ABB RAPID module: P61.mod

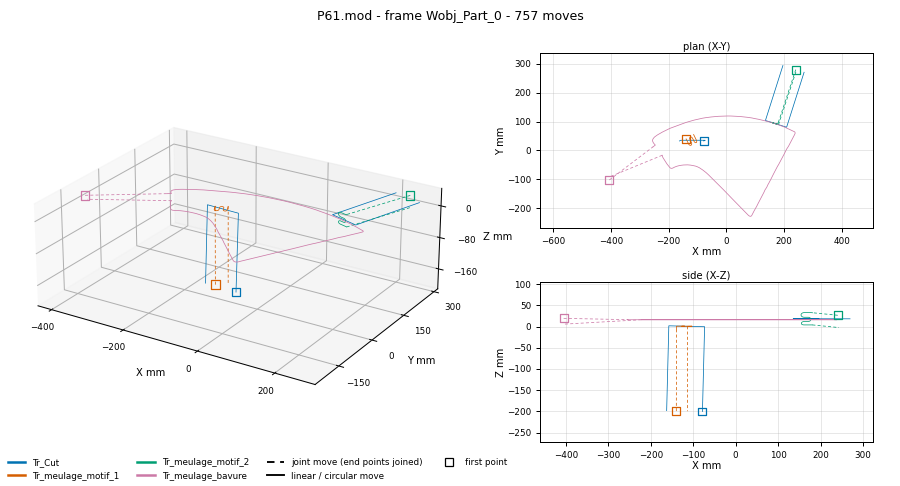
[picture p0: tool path of P61.mod in frame Wobj_Part_0, 757 of 767 moves have a stored position in this frame; points joined in program order, loops and branches not executed]
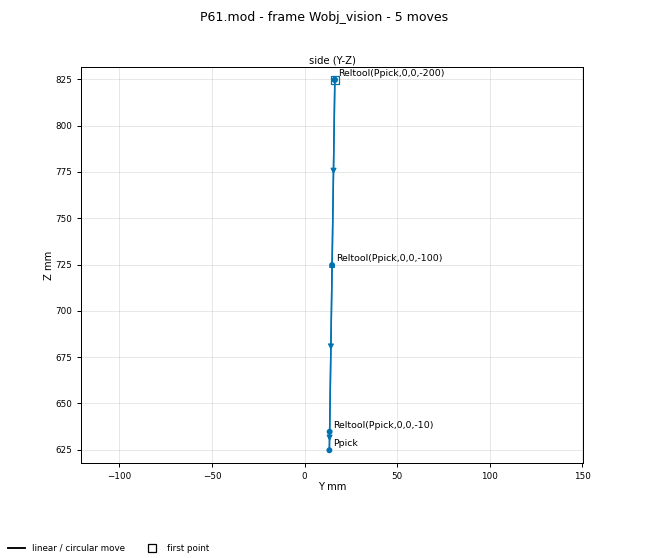
[picture p1: tool path of P61.mod in frame Wobj_vision, 5 of 767 moves have a stored position in this frame; points joined in program order, loops and branches not executed]
MODULE P61
	LOCAL CONST Speeddata vitesse_Tronconnage :=[10, 500, 0, 0];
	LOCAL CONST Robtarget Coupe_0 :=[[-120.4273984375,35.4203203125,0.733973022460938],[0.716031512015104,-0.00434153413134131,-0.698040250859739,0.00445343265621212],[0,0,0,0],[8.999999E+09,8.999999E+09,8.999999E+09,8.999999E+09,8.999999E+09,8.999999E+09]];
	LOCAL CONST Robtarget Coupe_1 :=[[167.499296875,93.7912890625,18.2855390625],[0.417597748453561,0.417256329208566,-0.570874027904049,-0.570624325179462],[0,0,0,0],[8.999999E+09,8.999999E+09,8.999999E+09,8.999999E+09,8.999999E+09,8.999999E+09]];
	LOCAL CONST Robtarget Tr_meulage_motif_1_App1 :=[[-139.92964037527,40.0496042134107,-199.309536992709],[-7.8362214742082E-08,0.00132363335464177,5.92023053405581E-05,0.999999122244526],[0,0,0,0],[8.999999E+09,8.999999E+09,8.999999E+09,8.999999E+09,8.999999E+09,8.999999E+09]];
	LOCAL CONST Robtarget Tr_meulage_motif_1_App2 :=[[-139.426660143764,40.072101109108,-9.31020408657393],[-7.8362214742082E-08,0.00132363335464177,5.92023053405581E-05,0.999999122244526],[0,0,0,0],[8.999999E+09,8.999999E+09,8.999999E+09,8.999999E+09,8.999999E+09,8.999999E+09]];
	LOCAL CONST Robtarget Tr_meulage_motif_1_P0 :=[[-139.4001875,40.07328515625,0.689760803222656],[-7.8362214742082E-08,0.00132363335464177,5.92023053405581E-05,0.999999122244526],[0,0,0,0],[8.999999E+09,8.999999E+09,8.999999E+09,8.999999E+09,8.999999E+09,8.999999E+09]];
	LOCAL CONST Robtarget Tr_meulage_motif_1_P1 :=[[-138.96090625,39.1750078125,0.700619750976562],[-7.8362214742082E-08,0.00132363335464177,5.92023053405581E-05,0.999999122244526],[0,0,0,0],[8.999999E+09,8.999999E+09,8.999999E+09,8.999999E+09,8.999999E+09,8.999999E+09]];
	LOCAL CONST Robtarget Tr_meulage_motif_1_P2 :=[[-138.521609375,38.27673046875,0.711478759765625],[-7.8362214742082E-08,0.00132363335464177,5.92023053405581E-05,0.999999122244526],[0,0,0,0],[8.999999E+09,8.999999E+09,8.999999E+09,8.999999E+09,8.999999E+09,8.999999E+09]];
	LOCAL CONST Robtarget Tr_meulage_motif_1_P3 :=[[-138.0823125,37.378453125,0.722337707519531],[-7.8362214742082E-08,0.00132363335464177,5.92023053405581E-05,0.999999122244526],[0,0,0,0],[8.999999E+09,8.999999E+09,8.999999E+09,8.999999E+09,8.999999E+09,8.999999E+09]];
	LOCAL CONST Robtarget Tr_meulage_motif_1_P4 :=[[-137.643015625,36.480171875,0.733196716308594],[-7.8362214742082E-08,0.00132363335464177,5.92023053405581E-05,0.999999122244526],[0,0,0,0],[8.999999E+09,8.999999E+09,8.999999E+09,8.999999E+09,8.999999E+09,8.999999E+09]];
	LOCAL CONST Robtarget Tr_meulage_motif_1_P5 :=[[-137.203734375,35.58189453125,0.744055725097656],[-7.8362214742082E-08,0.00132363335464177,5.92023053405581E-05,0.999999122244526],[0,0,0,0],[8.999999E+09,8.999999E+09,8.999999E+09,8.999999E+09,8.999999E+09,8.999999E+09]];
	LOCAL CONST Robtarget Tr_meulage_motif_1_P6 :=[[-136.7644375,34.6836171875,0.754914672851563],[-7.8362214742082E-08,0.00132363335464177,5.92023053405581E-05,0.999999122244526],[0,0,0,0],[8.999999E+09,8.999999E+09,8.999999E+09,8.999999E+09,8.999999E+09,8.999999E+09]];
	LOCAL CONST Robtarget Tr_meulage_motif_1_P7 :=[[-136.325140625,33.78533984375,0.765773681640625],[-7.8362214742082E-08,0.00132363335464177,5.92023053405581E-05,0.999999122244526],[0,0,0,0],[8.999999E+09,8.999999E+09,8.999999E+09,8.999999E+09,8.999999E+09,8.999999E+09]];
	LOCAL CONST Robtarget Tr_meulage_motif_1_P8 :=[[-135.88584375,32.88705859375,0.776632629394531],[-7.8362214742082E-08,0.00132363335464177,5.92023053405581E-05,0.999999122244526],[0,0,0,0],[8.999999E+09,8.999999E+09,8.999999E+09,8.999999E+09,8.999999E+09,8.999999E+09]];
	LOCAL CONST Robtarget Tr_meulage_motif_1_P9 :=[[-135.4465625,31.98878125,0.787491638183594],[-7.8362214742082E-08,0.00132363335464177,5.92023053405581E-05,0.999999122244526],[0,0,0,0],[8.999999E+09,8.999999E+09,8.999999E+09,8.999999E+09,8.999999E+09,8.999999E+09]];
	LOCAL CONST Robtarget Tr_meulage_motif_1_P10 :=[[-135.007265625,31.09050390625,0.7983505859375],[-7.8362214742082E-08,0.00132363335464177,5.92023053405581E-05,0.999999122244526],[0,0,0,0],[8.999999E+09,8.999999E+09,8.999999E+09,8.999999E+09,8.999999E+09,8.999999E+09]];
	LOCAL CONST Robtarget Tr_meulage_motif_1_P11 :=[[-134.56796875,30.192224609375,0.809209594726563],[-7.8362214742082E-08,0.00132363335464177,5.92023053405581E-05,0.999999122244526],[0,0,0,0],[8.999999E+09,8.999999E+09,8.999999E+09,8.999999E+09,8.999999E+09,8.999999E+09]];
	LOCAL CONST Robtarget Tr_meulage_motif_1_P12 :=[[-134.128671875,29.293947265625,0.820068603515625],[-7.8362214742082E-08,0.00132363335464177,5.92023053405581E-05,0.999999122244526],[0,0,0,0],[8.999999E+09,8.999999E+09,8.999999E+09,8.999999E+09,8.999999E+09,8.999999E+09]];
	LOCAL CONST Robtarget Tr_meulage_motif_1_P13 :=[[-133.689390625,28.39566796875,0.830927551269531],[-7.8362214742082E-08,0.00132363335464177,5.92023053405581E-05,0.999999122244526],[0,0,0,0],[8.999999E+09,8.999999E+09,8.999999E+09,8.999999E+09,8.999999E+09,8.999999E+09]];
	LOCAL CONST Robtarget Tr_meulage_motif_1_P14 :=[[-133.25009375,27.497390625,0.841786560058594],[-7.8362214742082E-08,0.00132363335464177,5.92023053405581E-05,0.999999122244526],[0,0,0,0],[8.999999E+09,8.999999E+09,8.999999E+09,8.999999E+09,8.999999E+09,8.999999E+09]];
	LOCAL CONST Robtarget Tr_meulage_motif_1_P15 :=[[-132.810796875,26.599111328125,0.8526455078125],[-7.8362214742082E-08,0.00132363335464177,5.92023053405581E-05,0.999999122244526],[0,0,0,0],[8.999999E+09,8.999999E+09,8.999999E+09,8.999999E+09,8.999999E+09,8.999999E+09]];
	LOCAL CONST Robtarget Tr_meulage_motif_1_P16 :=[[-132.371515625,25.700833984375,0.863504516601562],[-7.8362214742082E-08,0.00132363335464177,5.92023053405581E-05,0.999999122244526],[0,0,0,0],[8.999999E+09,8.999999E+09,8.999999E+09,8.999999E+09,8.999999E+09,8.999999E+09]];
	LOCAL CONST Robtarget Tr_meulage_motif_1_P17 :=[[-131.93221875,24.8025546875,0.874363525390625],[-7.8362214742082E-08,0.00132363335464177,5.92023053405581E-05,0.999999122244526],[0,0,0,0],[8.999999E+09,8.999999E+09,8.999999E+09,8.999999E+09,8.999999E+09,8.999999E+09]];
	LOCAL CONST Robtarget Tr_meulage_motif_1_P18 :=[[-131.492921875,23.90427734375,0.885222473144531],[-7.8362214742082E-08,0.00132363335464177,5.92023053405581E-05,0.999999122244526],[0,0,0,0],[8.999999E+09,8.999999E+09,8.999999E+09,8.999999E+09,8.999999E+09,8.999999E+09]];
	LOCAL CONST Robtarget Tr_meulage_motif_1_P19 :=[[-131.0536328125,23.005998046875,0.896081481933594],[-7.8362214742082E-08,0.00132363335464177,5.92023053405581E-05,0.999999122244526],[0,0,0,0],[8.999999E+09,8.999999E+09,8.999999E+09,8.999999E+09,8.999999E+09,8.999999E+09]];
	LOCAL CONST Robtarget Tr_meulage_motif_1_P20 :=[[-130.6143359375,22.107720703125,0.9069404296875],[-7.8362214742082E-08,0.00132363335464177,5.92023053405581E-05,0.999999122244526],[0,0,0,0],[8.999999E+09,8.999999E+09,8.999999E+09,8.999999E+09,8.999999E+09,8.999999E+09]];
	LOCAL CONST Robtarget Tr_meulage_motif_1_P21 :=[[-130.0789609375,21.264701171875,0.917042663574219],[-7.8362214742082E-08,0.00132363335464177,5.92023053405581E-05,0.999999122244526],[0,0,0,0],[8.999999E+09,8.999999E+09,8.999999E+09,8.999999E+09,8.999999E+09,8.999999E+09]];
	LOCAL CONST Robtarget Tr_meulage_motif_1_P22 :=[[-129.473453125,20.507244140625,0.926029846191406],[-7.8362214742082E-08,0.00132363335464177,5.92023053405581E-05,0.999999122244526],[0,0,0,0],[8.999999E+09,8.999999E+09,8.999999E+09,8.999999E+09,8.999999E+09,8.999999E+09]];
	LOCAL CONST Robtarget Tr_meulage_motif_1_P23 :=[[-128.8546484375,19.860673828125,0.9336279296875],[-7.8362214742082E-08,0.00132363335464177,5.92023053405581E-05,0.999999122244526],[0,0,0,0],[8.999999E+09,8.999999E+09,8.999999E+09,8.999999E+09,8.999999E+09,8.999999E+09]];
	LOCAL CONST Robtarget Tr_meulage_motif_1_P24 :=[[-128.2773203125,19.3082265625,0.940084838867188],[-7.8362214742082E-08,0.00132363335464177,5.92023053405581E-05,0.999999122244526],[0,0,0,0],[8.999999E+09,8.999999E+09,8.999999E+09,8.999999E+09,8.999999E+09,8.999999E+09]];
	LOCAL CONST Robtarget Tr_meulage_motif_1_P25 :=[[-127.240140625,18.589798828125,0.948275268554687],[-7.8362214742082E-08,0.00132363335464177,5.92023053405581E-05,0.999999122244526],[0,0,0,0],[8.999999E+09,8.999999E+09,8.999999E+09,8.999999E+09,8.999999E+09,8.999999E+09]];
	LOCAL CONST Robtarget Tr_meulage_motif_1_P26 :=[[-126.028875,18.042408203125,0.954212341308594],[-7.8362214742082E-08,0.00132363335464177,5.92023053405581E-05,0.999999122244526],[0,0,0,0],[8.999999E+09,8.999999E+09,8.999999E+09,8.999999E+09,8.999999E+09,8.999999E+09]];
	LOCAL CONST Robtarget Tr_meulage_motif_1_P27 :=[[-124.7367109375,17.73071484375,0.957158752441406],[-7.8362214742082E-08,0.00132363335464177,5.92023053405581E-05,0.999999122244526],[0,0,0,0],[8.999999E+09,8.999999E+09,8.999999E+09,8.999999E+09,8.999999E+09,8.999999E+09]];
	LOCAL CONST Robtarget Tr_meulage_motif_1_P28 :=[[-123.519546875,17.782501953125,0.955637145996094],[-7.8362214742082E-08,0.00132363335464177,5.92023053405581E-05,0.999999122244526],[0,0,0,0],[8.999999E+09,8.999999E+09,8.999999E+09,8.999999E+09,8.999999E+09,8.999999E+09]];
	LOCAL CONST Robtarget Tr_meulage_motif_1_P29 :=[[-122.8824375,18.063896484375,0.951677001953125],[-7.8362214742082E-08,0.00132363335464177,5.92023053405581E-05,0.999999122244526],[0,0,0,0],[8.999999E+09,8.999999E+09,8.999999E+09,8.999999E+09,8.999999E+09,8.999999E+09]];
	LOCAL CONST Robtarget Tr_meulage_motif_1_P30 :=[[-122.28840625,18.3543515625,0.947635192871094],[-7.8362214742082E-08,0.00132363335464177,5.92023053405581E-05,0.999999122244526],[0,0,0,0],[8.999999E+09,8.999999E+09,8.999999E+09,8.999999E+09,8.999999E+09,8.999999E+09]];
	LOCAL CONST Robtarget Tr_meulage_motif_1_P31 :=[[-121.718625,18.69403125,0.942998474121094],[-7.8362214742082E-08,0.00132363335464177,5.92023053405581E-05,0.999999122244526],[0,0,0,0],[8.999999E+09,8.999999E+09,8.999999E+09,8.999999E+09,8.999999E+09,8.999999E+09]];
	LOCAL CONST Robtarget Tr_meulage_motif_1_P32 :=[[-120.9477421875,19.625513671875,0.930854064941406],[-7.8362214742082E-08,0.00132363335464177,5.92023053405581E-05,0.999999122244526],[0,0,0,0],[8.999999E+09,8.999999E+09,8.999999E+09,8.999999E+09,8.999999E+09,8.999999E+09]];
	LOCAL CONST Robtarget Tr_meulage_motif_1_P33 :=[[-120.4197578125,20.837162109375,0.915399108886719],[-7.8362214742082E-08,0.00132363335464177,5.92023053405581E-05,0.999999122244526],[0,0,0,0],[8.999999E+09,8.999999E+09,8.999999E+09,8.999999E+09,8.999999E+09,8.999999E+09]];
	LOCAL CONST Robtarget Tr_meulage_motif_1_P34 :=[[-120.1247109375,22.12055078125,0.899219604492188],[-7.8362214742082E-08,0.00132363335464177,5.92023053405581E-05,0.999999122244526],[0,0,0,0],[8.999999E+09,8.999999E+09,8.999999E+09,8.999999E+09,8.999999E+09,8.999999E+09]];
	LOCAL CONST Robtarget Tr_meulage_motif_1_P35 :=[[-120.07103125,22.9115859375,0.889339538574219],[-7.8362214742082E-08,0.00132363335464177,5.92023053405581E-05,0.999999122244526],[0,0,0,0],[8.999999E+09,8.999999E+09,8.999999E+09,8.999999E+09,8.999999E+09,8.999999E+09]];
	LOCAL CONST Robtarget Tr_meulage_motif_1_P36 :=[[-120.141828125,24.166080078125,0.873783142089844],[-7.8362214742082E-08,0.00132363335464177,5.92023053405581E-05,0.999999122244526],[0,0,0,0],[8.999999E+09,8.999999E+09,8.999999E+09,8.999999E+09,8.999999E+09,8.999999E+09]];
	LOCAL CONST Robtarget Tr_meulage_motif_1_P37 :=[[-120.275796875,25.04115625,0.862992736816406],[-7.8362214742082E-08,0.00132363335464177,5.92023053405581E-05,0.999999122244526],[0,0,0,0],[8.999999E+09,8.999999E+09,8.999999E+09,8.999999E+09,8.999999E+09,8.999999E+09]];
	LOCAL CONST Robtarget Tr_meulage_motif_1_P38 :=[[-120.5015390625,25.968166015625,0.851622375488281],[-7.8362214742082E-08,0.00132363335464177,5.92023053405581E-05,0.999999122244526],[0,0,0,0],[8.999999E+09,8.999999E+09,8.999999E+09,8.999999E+09,8.999999E+09,8.999999E+09]];
	LOCAL CONST Robtarget Tr_meulage_motif_1_P39 :=[[-120.835171875,26.89758203125,0.840299865722656],[-7.8362214742082E-08,0.00132363335464177,5.92023053405581E-05,0.999999122244526],[0,0,0,0],[8.999999E+09,8.999999E+09,8.999999E+09,8.999999E+09,8.999999E+09,8.999999E+09]];
	LOCAL CONST Robtarget Tr_meulage_motif_1_P40 :=[[-121.1718515625,27.8377578125,0.828845642089844],[-7.8362214742082E-08,0.00132363335464177,5.92023053405581E-05,0.999999122244526],[0,0,0,0],[8.999999E+09,8.999999E+09,8.999999E+09,8.999999E+09,8.999999E+09,8.999999E+09]];
	LOCAL CONST Robtarget Tr_meulage_motif_1_P41 :=[[-121.611140625,28.73603515625,0.817986633300781],[-7.8362214742082E-08,0.00132363335464177,5.92023053405581E-05,0.999999122244526],[0,0,0,0],[8.999999E+09,8.999999E+09,8.999999E+09,8.999999E+09,8.999999E+09,8.999999E+09]];
	LOCAL CONST Robtarget Tr_meulage_motif_1_P42 :=[[-122.0504375,29.634314453125,0.807127685546875],[-7.8362214742082E-08,0.00132363335464177,5.92023053405581E-05,0.999999122244526],[0,0,0,0],[8.999999E+09,8.999999E+09,8.999999E+09,8.999999E+09,8.999999E+09,8.999999E+09]];
	LOCAL CONST Robtarget Tr_meulage_motif_1_P43 :=[[-122.4897265625,30.532591796875,0.796268676757813],[-7.8362214742082E-08,0.00132363335464177,5.92023053405581E-05,0.999999122244526],[0,0,0,0],[8.999999E+09,8.999999E+09,8.999999E+09,8.999999E+09,8.999999E+09,8.999999E+09]];
	LOCAL CONST Robtarget Tr_meulage_motif_1_P44 :=[[-122.9290234375,31.43087109375,0.785409729003906],[-7.8362214742082E-08,0.00132363335464177,5.92023053405581E-05,0.999999122244526],[0,0,0,0],[8.999999E+09,8.999999E+09,8.999999E+09,8.999999E+09,8.999999E+09,8.999999E+09]];
	LOCAL CONST Robtarget Tr_meulage_motif_1_P45 :=[[-123.3683125,32.3291484375,0.774550720214844],[-7.8362214742082E-08,0.00132363335464177,5.92023053405581E-05,0.999999122244526],[0,0,0,0],[8.999999E+09,8.999999E+09,8.999999E+09,8.999999E+09,8.999999E+09,8.999999E+09]];
	LOCAL CONST Robtarget Tr_meulage_motif_1_P46 :=[[-123.807609375,33.22742578125,0.763691711425781],[-7.8362214742082E-08,0.00132363335464177,5.92023053405581E-05,0.999999122244526],[0,0,0,0],[8.999999E+09,8.999999E+09,8.999999E+09,8.999999E+09,8.999999E+09,8.999999E+09]];
	LOCAL CONST Robtarget Tr_meulage_motif_1_P47 :=[[-124.2468984375,34.12570703125,0.752832763671875],[-7.8362214742082E-08,0.00132363335464177,5.92023053405581E-05,0.999999122244526],[0,0,0,0],[8.999999E+09,8.999999E+09,8.999999E+09,8.999999E+09,8.999999E+09,8.999999E+09]];
	LOCAL CONST Robtarget Tr_meulage_motif_1_P48 :=[[-124.6861953125,35.023984375,0.741973754882812],[-7.8362214742082E-08,0.00132363335464177,5.92023053405581E-05,0.999999122244526],[0,0,0,0],[8.999999E+09,8.999999E+09,8.999999E+09,8.999999E+09,8.999999E+09,8.999999E+09]];
	LOCAL CONST Robtarget Tr_meulage_motif_1_P49 :=[[-125.125484375,35.92226171875,0.731114807128906],[-7.8362214742082E-08,0.00132363335464177,5.92023053405581E-05,0.999999122244526],[0,0,0,0],[8.999999E+09,8.999999E+09,8.999999E+09,8.999999E+09,8.999999E+09,8.999999E+09]];
	LOCAL CONST Robtarget Tr_meulage_motif_1_P50 :=[[-125.56478125,36.8205390625,0.720255798339844],[-7.8362214742082E-08,0.00132363335464177,5.92023053405581E-05,0.999999122244526],[0,0,0,0],[8.999999E+09,8.999999E+09,8.999999E+09,8.999999E+09,8.999999E+09,8.999999E+09]];
	LOCAL CONST Robtarget Tr_meulage_motif_1_P51 :=[[-126.0040703125,37.7188203125,0.709396789550781],[-7.8362214742082E-08,0.00132363335464177,5.92023053405581E-05,0.999999122244526],[0,0,0,0],[8.999999E+09,8.999999E+09,8.999999E+09,8.999999E+09,8.999999E+09,8.999999E+09]];
	LOCAL CONST Robtarget Tr_meulage_motif_1_P52 :=[[-126.443359375,38.61709765625,0.698537841796875],[-7.8362214742082E-08,0.00132363335464177,5.92023053405581E-05,0.999999122244526],[0,0,0,0],[8.999999E+09,8.999999E+09,8.999999E+09,8.999999E+09,8.999999E+09,8.999999E+09]];
	LOCAL CONST Robtarget Tr_meulage_motif_1_P53 :=[[-126.7800390625,39.5572734375,0.687083618164062],[-7.8362214742082E-08,0.00132363335464177,5.92023053405581E-05,0.999999122244526],[0,0,0,0],[8.999999E+09,8.999999E+09,8.999999E+09,8.999999E+09,8.999999E+09,8.999999E+09]];
	LOCAL CONST Robtarget Tr_meulage_motif_1_P54 :=[[-127.006109375,40.5002578125,0.675514770507813],[-7.8362214742082E-08,0.00132363335464177,5.92023053405581E-05,0.999999122244526],[0,0,0,0],[8.999999E+09,8.999999E+09,8.999999E+09,8.999999E+09,8.999999E+09,8.999999E+09]];
	LOCAL CONST Robtarget Tr_meulage_motif_1_P55 :=[[-127.1364921875,41.38564453125,0.664593505859375],[-7.8362214742082E-08,0.00132363335464177,5.92023053405581E-05,0.999999122244526],[0,0,0,0],[8.999999E+09,8.999999E+09,8.999999E+09,8.999999E+09,8.999999E+09,8.999999E+09]];
	LOCAL CONST Robtarget Tr_meulage_motif_1_P56 :=[[-127.1758125,42.15837109375,0.655008239746094],[-7.8362214742082E-08,0.00132363335464177,5.92023053405581E-05,0.999999122244526],[0,0,0,0],[8.999999E+09,8.999999E+09,8.999999E+09,8.999999E+09,8.999999E+09,8.999999E+09]];
	LOCAL CONST Robtarget Tr_meulage_motif_1_P57 :=[[-127.0350703125,43.37862890625,0.639725280761719],[-7.8362214742082E-08,0.00132363335464177,5.92023053405581E-05,0.999999122244526],[0,0,0,0],[8.999999E+09,8.999999E+09,8.999999E+09,8.999999E+09,8.999999E+09,8.999999E+09]];
	LOCAL CONST Robtarget Tr_meulage_motif_1_P58 :=[[-126.62103125,44.58499609375,0.624418212890625],[-7.8362214742082E-08,0.00132363335464177,5.92023053405581E-05,0.999999122244526],[0,0,0,0],[8.999999E+09,8.999999E+09,8.999999E+09,8.999999E+09,8.999999E+09,8.999999E+09]];
	LOCAL CONST Robtarget Tr_meulage_motif_1_P59 :=[[-125.91634375,45.525015625,0.61221533203125],[-7.8362214742082E-08,0.00132363335464177,5.92023053405581E-05,0.999999122244526],[0,0,0,0],[8.999999E+09,8.999999E+09,8.999999E+09,8.999999E+09,8.999999E+09,8.999999E+09]];
	LOCAL CONST Robtarget Tr_meulage_motif_1_P60 :=[[-125.374765625,45.9955,0.605971557617187],[-7.8362214742082E-08,0.00132363335464177,5.92023053405581E-05,0.999999122244526],[0,0,0,0],[8.999999E+09,8.999999E+09,8.999999E+09,8.999999E+09,8.999999E+09,8.999999E+09]];
	LOCAL CONST Robtarget Tr_meulage_motif_1_P61 :=[[-124.71109375,46.3910703125,0.60057177734375],[-7.8362214742082E-08,0.00132363335464177,5.92023053405581E-05,0.999999122244526],[0,0,0,0],[8.999999E+09,8.999999E+09,8.999999E+09,8.999999E+09,8.999999E+09,8.999999E+09]];
	LOCAL CONST Robtarget Tr_meulage_motif_1_P62 :=[[-123.9900703125,46.669109375,0.596592895507812],[-7.8362214742082E-08,0.00132363335464177,5.92023053405581E-05,0.999999122244526],[0,0,0,0],[8.999999E+09,8.999999E+09,8.999999E+09,8.999999E+09,8.999999E+09,8.999999E+09]];
	LOCAL CONST Robtarget Tr_meulage_motif_1_P63 :=[[-122.81015625,46.779,0.594375244140625],[-7.8362214742082E-08,0.00132363335464177,5.92023053405581E-05,0.999999122244526],[0,0,0,0],[8.999999E+09,8.999999E+09,8.999999E+09,8.999999E+09,8.999999E+09,8.999999E+09]];
	LOCAL CONST Robtarget Tr_meulage_motif_1_P64 :=[[-122.1020078125,46.66409375,0.595294372558594],[-7.8362214742082E-08,0.00132363335464177,5.92023053405581E-05,0.999999122244526],[0,0,0,0],[8.999999E+09,8.999999E+09,8.999999E+09,8.999999E+09,8.999999E+09,8.999999E+09]];
	LOCAL CONST Robtarget Tr_meulage_motif_1_P65 :=[[-120.9153515625,46.25687890625,0.599505187988281],[-7.8362214742082E-08,0.00132363335464177,5.92023053405581E-05,0.999999122244526],[0,0,0,0],[8.999999E+09,8.999999E+09,8.999999E+09,8.999999E+09,8.999999E+09,8.999999E+09]];
	LOCAL CONST Robtarget Tr_meulage_motif_1_P66 :=[[-120.285875,45.9127578125,0.603332763671875],[-7.8362214742082E-08,0.00132363335464177,5.92023053405581E-05,0.999999122244526],[0,0,0,0],[8.999999E+09,8.999999E+09,8.999999E+09,8.999999E+09,8.999999E+09,8.999999E+09]];
	LOCAL CONST Robtarget Tr_meulage_motif_1_P67 :=[[-119.306,45.14755859375,0.612146423339844],[-7.8362214742082E-08,0.00132363335464177,5.92023053405581E-05,0.999999122244526],[0,0,0,0],[8.999999E+09,8.999999E+09,8.999999E+09,8.999999E+09,8.999999E+09,8.999999E+09]];
	LOCAL CONST Robtarget Tr_meulage_motif_1_P68 :=[[-118.677859375,44.53574609375,0.619305297851563],[-7.8362214742082E-08,0.00132363335464177,5.92023053405581E-05,0.999999122244526],[0,0,0,0],[8.999999E+09,8.999999E+09,8.999999E+09,8.999999E+09,8.999999E+09,8.999999E+09]];
	LOCAL CONST Robtarget Tr_meulage_motif_1_P69 :=[[-118.0847578125,43.78836328125,0.628176086425781],[-7.8362214742082E-08,0.00132363335464177,5.92023053405581E-05,0.999999122244526],[0,0,0,0],[8.999999E+09,8.999999E+09,8.999999E+09,8.999999E+09,8.999999E+09,8.999999E+09]];
	LOCAL CONST Robtarget Tr_meulage_motif_1_P70 :=[[-117.5560078125,42.95434765625,0.638171081542969],[-7.8362214742082E-08,0.00132363335464177,5.92023053405581E-05,0.999999122244526],[0,0,0,0],[8.999999E+09,8.999999E+09,8.999999E+09,8.999999E+09,8.999999E+09,8.999999E+09]];
	LOCAL CONST Robtarget Tr_meulage_motif_1_P71 :=[[-117.0206328125,42.111328125,0.648273315429687],[-7.8362214742082E-08,0.00132363335464177,5.92023053405581E-05,0.999999122244526],[0,0,0,0],[8.999999E+09,8.999999E+09,8.999999E+09,8.999999E+09,8.999999E+09,8.999999E+09]];
	LOCAL CONST Robtarget Tr_meulage_motif_1_P72 :=[[-116.58134375,41.21305078125,0.65913232421875],[-7.8362214742082E-08,0.00132363335464177,5.92023053405581E-05,0.999999122244526],[0,0,0,0],[8.999999E+09,8.999999E+09,8.999999E+09,8.999999E+09,8.999999E+09,8.999999E+09]];
	LOCAL CONST Robtarget Tr_meulage_motif_1_P73 :=[[-116.142046875,40.31476953125,0.669991333007813],[-7.8362214742082E-08,0.00132363335464177,5.92023053405581E-05,0.999999122244526],[0,0,0,0],[8.999999E+09,8.999999E+09,8.999999E+09,8.999999E+09,8.999999E+09,8.999999E+09]];
	LOCAL CONST Robtarget Tr_meulage_motif_1_P74 :=[[-115.7027578125,39.4164921875,0.680850280761719],[-7.8362214742082E-08,0.00132363335464177,5.92023053405581E-05,0.999999122244526],[0,0,0,0],[8.999999E+09,8.999999E+09,8.999999E+09,8.999999E+09,8.999999E+09,8.999999E+09]];
	LOCAL CONST Robtarget Tr_meulage_motif_1_P75 :=[[-115.2634609375,38.51821484375,0.691709289550781],[-7.8362214742082E-08,0.00132363335464177,5.92023053405581E-05,0.999999122244526],[0,0,0,0],[8.999999E+09,8.999999E+09,8.999999E+09,8.999999E+09,8.999999E+09,8.999999E+09]];
	LOCAL CONST Robtarget Tr_meulage_motif_1_P76 :=[[-114.824171875,37.6199375,0.702568237304688],[-7.8362214742082E-08,0.00132363335464177,5.92023053405581E-05,0.999999122244526],[0,0,0,0],[8.999999E+09,8.999999E+09,8.999999E+09,8.999999E+09,8.999999E+09,8.999999E+09]];
	LOCAL CONST Robtarget Tr_meulage_motif_1_P77 :=[[-114.384875,36.72165625,0.71342724609375],[-7.8362214742082E-08,0.00132363335464177,5.92023053405581E-05,0.999999122244526],[0,0,0,0],[8.999999E+09,8.999999E+09,8.999999E+09,8.999999E+09,8.999999E+09,8.999999E+09]];
	LOCAL CONST Robtarget Tr_meulage_motif_1_P78 :=[[-113.9455859375,35.82337890625,0.724286193847656],[-7.8362214742082E-08,0.00132363335464177,5.92023053405581E-05,0.999999122244526],[0,0,0,0],[8.999999E+09,8.999999E+09,8.999999E+09,8.999999E+09,8.999999E+09,8.999999E+09]];
	LOCAL CONST Robtarget Tr_meulage_motif_1_P79 :=[[-113.5062890625,34.9251015625,0.735145202636719],[-7.8362214742082E-08,0.00132363335464177,5.92023053405581E-05,0.999999122244526],[0,0,0,0],[8.999999E+09,8.999999E+09,8.999999E+09,8.999999E+09,8.999999E+09,8.999999E+09]];
	LOCAL CONST Robtarget Tr_meulage_motif_1_P80 :=[[-113.067,34.02682421875,0.746004211425781],[-7.8362214742082E-08,0.00132363335464177,5.92023053405581E-05,0.999999122244526],[0,0,0,0],[8.999999E+09,8.999999E+09,8.999999E+09,8.999999E+09,8.999999E+09,8.999999E+09]];
	LOCAL CONST Robtarget Tr_meulage_motif_1_P81 :=[[-112.627703125,33.12854296875,0.756863159179687],[-7.8362214742082E-08,0.00132363335464177,5.92023053405581E-05,0.999999122244526],[0,0,0,0],[8.999999E+09,8.999999E+09,8.999999E+09,8.999999E+09,8.999999E+09,8.999999E+09]];
	LOCAL CONST Robtarget Tr_meulage_motif_1_P82 :=[[-112.1884140625,32.230265625,0.76772216796875],[-7.8362214742082E-08,0.00132363335464177,5.92023053405581E-05,0.999999122244526],[0,0,0,0],[8.999999E+09,8.999999E+09,8.999999E+09,8.999999E+09,8.999999E+09,8.999999E+09]];
	LOCAL CONST Robtarget Tr_meulage_motif_1_P83 :=[[-111.7491171875,31.33198828125,0.778581115722656],[-7.8362214742082E-08,0.00132363335464177,5.92023053405581E-05,0.999999122244526],[0,0,0,0],[8.999999E+09,8.999999E+09,8.999999E+09,8.999999E+09,8.999999E+09,8.999999E+09]];
	LOCAL CONST Robtarget Tr_meulage_motif_1_P84 :=[[-111.2137421875,30.48896875,0.788683349609375],[-7.8362214742082E-08,0.00132363335464177,5.92023053405581E-05,0.999999122244526],[0,0,0,0],[8.999999E+09,8.999999E+09,8.999999E+09,8.999999E+09,8.999999E+09,8.999999E+09]];
	LOCAL CONST Robtarget Tr_meulage_motif_1_P85 :=[[-110.608234375,29.73151171875,0.797670532226562],[-7.8362214742082E-08,0.00132363335464177,5.92023053405581E-05,0.999999122244526],[0,0,0,0],[8.999999E+09,8.999999E+09,8.999999E+09,8.999999E+09,8.999999E+09,8.999999E+09]];
	LOCAL CONST Robtarget Tr_meulage_motif_1_P86 :=[[-109.9894296875,29.08494140625,0.805268615722656],[-7.8362214742082E-08,0.00132363335464177,5.92023053405581E-05,0.999999122244526],[0,0,0,0],[8.999999E+09,8.999999E+09,8.999999E+09,8.999999E+09,8.999999E+09,8.999999E+09]];
	LOCAL CONST Robtarget Tr_meulage_motif_1_P87 :=[[-109.4121015625,28.532494140625,0.811725524902344],[-7.8362214742082E-08,0.00132363335464177,5.92023053405581E-05,0.999999122244526],[0,0,0,0],[8.999999E+09,8.999999E+09,8.999999E+09,8.999999E+09,8.999999E+09,8.999999E+09]];
	LOCAL CONST Robtarget Tr_meulage_motif_1_P88 :=[[-108.374921875,27.81406640625,0.819916015625],[-7.8362214742082E-08,0.00132363335464177,5.92023053405581E-05,0.999999122244526],[0,0,0,0],[8.999999E+09,8.999999E+09,8.999999E+09,8.999999E+09,8.999999E+09,8.999999E+09]];
	LOCAL CONST Robtarget Tr_meulage_motif_1_P89 :=[[-107.16365625,27.26667578125,0.825853088378906],[-7.8362214742082E-08,0.00132363335464177,5.92023053405581E-05,0.999999122244526],[0,0,0,0],[8.999999E+09,8.999999E+09,8.999999E+09,8.999999E+09,8.999999E+09,8.999999E+09]];
	LOCAL CONST Robtarget Tr_meulage_motif_1_P90 :=[[-105.8764375,27.058552734375,0.827514526367187],[-7.8362214742082E-08,0.00132363335464177,5.92023053405581E-05,0.999999122244526],[0,0,0,0],[8.999999E+09,8.999999E+09,8.999999E+09,8.999999E+09,8.999999E+09,8.999999E+09]];
	LOCAL CONST Robtarget Tr_meulage_motif_1_P91 :=[[-104.7729765625,27.249388671875,0.824344848632813],[-7.8362214742082E-08,0.00132363335464177,5.92023053405581E-05,0.999999122244526],[0,0,0,0],[8.999999E+09,8.999999E+09,8.999999E+09,8.999999E+09,8.999999E+09,8.999999E+09]];
	LOCAL CONST Robtarget Tr_meulage_motif_1_P92 :=[[-104.2773125,27.557384765625,0.82015576171875],[-7.8362214742082E-08,0.00132363335464177,5.92023053405581E-05,0.999999122244526],[0,0,0,0],[8.999999E+09,8.999999E+09,8.999999E+09,8.999999E+09,8.999999E+09,8.999999E+09]];
	LOCAL CONST Robtarget Tr_meulage_motif_1_P93 :=[[-103.8999921875,27.737076171875,0.817648193359375],[-7.8362214742082E-08,0.00132363335464177,5.92023053405581E-05,0.999999122244526],[0,0,0,0],[8.999999E+09,8.999999E+09,8.999999E+09,8.999999E+09,8.999999E+09,8.999999E+09]];
	LOCAL CONST Robtarget Tr_meulage_motif_1_P94 :=[[-103.1883125,28.488166015625,0.807790771484375],[-7.8362214742082E-08,0.00132363335464177,5.92023053405581E-05,0.999999122244526],[0,0,0,0],[8.999999E+09,8.999999E+09,8.999999E+09,8.999999E+09,8.999999E+09,8.999999E+09]];
	LOCAL CONST Robtarget Tr_meulage_motif_1_P95 :=[[-102.7250078125,29.629576171875,0.79325634765625],[-7.8362214742082E-08,0.00132363335464177,5.92023053405581E-05,0.999999122244526],[0,0,0,0],[8.999999E+09,8.999999E+09,8.999999E+09,8.999999E+09,8.999999E+09,8.999999E+09]];
	LOCAL CONST Robtarget Tr_meulage_motif_1_P96 :=[[-102.613984375,30.36523828125,0.784023803710937],[-7.8362214742082E-08,0.00132363335464177,5.92023053405581E-05,0.999999122244526],[0,0,0,0],[8.999999E+09,8.999999E+09,8.999999E+09,8.999999E+09,8.999999E+09,8.999999E+09]];
	LOCAL CONST Robtarget Tr_meulage_motif_1_P97 :=[[-102.6340078125,31.613568359375,0.768507507324219],[-7.8362214742082E-08,0.00132363335464177,5.92023053405581E-05,0.999999122244526],[0,0,0,0],[8.999999E+09,8.999999E+09,8.999999E+09,8.999999E+09,8.999999E+09,8.999999E+09]];
	LOCAL CONST Robtarget Tr_meulage_motif_1_P98 :=[[-102.7679765625,32.48864453125,0.757717102050781],[-7.8362214742082E-08,0.00132363335464177,5.92023053405581E-05,0.999999122244526],[0,0,0,0],[8.999999E+09,8.999999E+09,8.999999E+09,8.999999E+09,8.999999E+09,8.999999E+09]];
	LOCAL CONST Robtarget Tr_meulage_motif_1_P99 :=[[-102.9937109375,33.41565234375,0.746346740722656],[-7.8362214742082E-08,0.00132363335464177,5.92023053405581E-05,0.999999122244526],[0,0,0,0],[8.999999E+09,8.999999E+09,8.999999E+09,8.999999E+09,8.999999E+09,8.999999E+09]];
	LOCAL CONST Robtarget Tr_meulage_motif_1_P100 :=[[-103.3273515625,34.3450703125,0.735024230957031],[-7.8362214742082E-08,0.00132363335464177,5.92023053405581E-05,0.999999122244526],[0,0,0,0],[8.999999E+09,8.999999E+09,8.999999E+09,8.999999E+09,8.999999E+09,8.999999E+09]];
	LOCAL CONST Robtarget Tr_meulage_motif_1_P101 :=[[-103.6640234375,35.28524609375,0.723570007324219],[-7.8362214742082E-08,0.00132363335464177,5.92023053405581E-05,0.999999122244526],[0,0,0,0],[8.999999E+09,8.999999E+09,8.999999E+09,8.999999E+09,8.999999E+09,8.999999E+09]];
	LOCAL CONST Robtarget Tr_meulage_motif_1_P102 :=[[-104.1033203125,36.1835234375,0.712710998535156],[-7.8362214742082E-08,0.00132363335464177,5.92023053405581E-05,0.999999122244526],[0,0,0,0],[8.999999E+09,8.999999E+09,8.999999E+09,8.999999E+09,8.999999E+09,8.999999E+09]];
	LOCAL CONST Robtarget Tr_meulage_motif_1_P103 :=[[-104.542609375,37.08180078125,0.70185205078125],[-7.8362214742082E-08,0.00132363335464177,5.92023053405581E-05,0.999999122244526],[0,0,0,0],[8.999999E+09,8.999999E+09,8.999999E+09,8.999999E+09,8.999999E+09,8.999999E+09]];
	LOCAL CONST Robtarget Tr_meulage_motif_1_P104 :=[[-104.98190625,37.98008203125,0.690993041992187],[-7.8362214742082E-08,0.00132363335464177,5.92023053405581E-05,0.999999122244526],[0,0,0,0],[8.999999E+09,8.999999E+09,8.999999E+09,8.999999E+09,8.999999E+09,8.999999E+09]];
	LOCAL CONST Robtarget Tr_meulage_motif_1_P105 :=[[-105.4211953125,38.878359375,0.680134094238281],[-7.8362214742082E-08,0.00132363335464177,5.92023053405581E-05,0.999999122244526],[0,0,0,0],[8.999999E+09,8.999999E+09,8.999999E+09,8.999999E+09,8.999999E+09,8.999999E+09]];
	LOCAL CONST Robtarget Tr_meulage_motif_1_P106 :=[[-105.8604921875,39.77663671875,0.669275085449219],[-7.8362214742082E-08,0.00132363335464177,5.92023053405581E-05,0.999999122244526],[0,0,0,0],[8.999999E+09,8.999999E+09,8.999999E+09,8.999999E+09,8.999999E+09,8.999999E+09]];
	LOCAL CONST Robtarget Tr_meulage_motif_1_P107 :=[[-106.29978125,40.6749140625,0.658416137695312],[-7.8362214742082E-08,0.00132363335464177,5.92023053405581E-05,0.999999122244526],[0,0,0,0],[8.999999E+09,8.999999E+09,8.999999E+09,8.999999E+09,8.999999E+09,8.999999E+09]];
	LOCAL CONST Robtarget Tr_meulage_motif_1_P108 :=[[-106.739078125,41.5731953125,0.64755712890625],[-7.8362214742082E-08,0.00132363335464177,5.92023053405581E-05,0.999999122244526],[0,0,0,0],[8.999999E+09,8.999999E+09,8.999999E+09,8.999999E+09,8.999999E+09,8.999999E+09]];
	LOCAL CONST Robtarget Tr_meulage_motif_1_P109 :=[[-107.1783671875,42.47147265625,0.636698120117188],[-7.8362214742082E-08,0.00132363335464177,5.92023053405581E-05,0.999999122244526],[0,0,0,0],[8.999999E+09,8.999999E+09,8.999999E+09,8.999999E+09,8.999999E+09,8.999999E+09]];
	LOCAL CONST Robtarget Tr_meulage_motif_1_P110 :=[[-107.6176640625,43.36975,0.625839172363281],[-7.8362214742082E-08,0.00132363335464177,5.92023053405581E-05,0.999999122244526],[0,0,0,0],[8.999999E+09,8.999999E+09,8.999999E+09,8.999999E+09,8.999999E+09,8.999999E+09]];
	LOCAL CONST Robtarget Tr_meulage_motif_1_P111 :=[[-108.056953125,44.26802734375,0.614980163574219],[-7.8362214742082E-08,0.00132363335464177,5.92023053405581E-05,0.999999122244526],[0,0,0,0],[8.999999E+09,8.999999E+09,8.999999E+09,8.999999E+09,8.999999E+09,8.999999E+09]];
	LOCAL CONST Robtarget Tr_meulage_motif_1_P112 :=[[-108.49625,45.16630859375,0.604121215820313],[-7.8362214742082E-08,0.00132363335464177,5.92023053405581E-05,0.999999122244526],[0,0,0,0],[8.999999E+09,8.999999E+09,8.999999E+09,8.999999E+09,8.999999E+09,8.999999E+09]];
	LOCAL CONST Robtarget Tr_meulage_motif_1_P113 :=[[-108.9355390625,46.0645859375,0.59326220703125],[-7.8362214742082E-08,0.00132363335464177,5.92023053405581E-05,0.999999122244526],[0,0,0,0],[8.999999E+09,8.999999E+09,8.999999E+09,8.999999E+09,8.999999E+09,8.999999E+09]];
	LOCAL CONST Robtarget Tr_meulage_motif_1_P114 :=[[-109.3748359375,46.96286328125,0.582403198242188],[-7.8362214742082E-08,0.00132363335464177,5.92023053405581E-05,0.999999122244526],[0,0,0,0],[8.999999E+09,8.999999E+09,8.999999E+09,8.999999E+09,8.999999E+09,8.999999E+09]];
	LOCAL CONST Robtarget Tr_meulage_motif_1_P115 :=[[-109.814125,47.861140625,0.571544250488281],[-7.8362214742082E-08,0.00132363335464177,5.92023053405581E-05,0.999999122244526],[0,0,0,0],[8.999999E+09,8.999999E+09,8.999999E+09,8.999999E+09,8.999999E+09,8.999999E+09]];
	LOCAL CONST Robtarget Tr_meulage_motif_1_P116 :=[[-110.253421875,48.759421875,0.560685241699219],[-7.8362214742082E-08,0.00132363335464177,5.92023053405581E-05,0.999999122244526],[0,0,0,0],[8.999999E+09,8.999999E+09,8.999999E+09,8.999999E+09,8.999999E+09,8.999999E+09]];
	LOCAL CONST Robtarget Tr_meulage_motif_1_P117 :=[[-110.6927109375,49.65769921875,0.549826293945312],[-7.8362214742082E-08,0.00132363335464177,5.92023053405581E-05,0.999999122244526],[0,0,0,0],[8.999999E+09,8.999999E+09,8.999999E+09,8.999999E+09,8.999999E+09,8.999999E+09]];
	LOCAL CONST Robtarget Tr_meulage_motif_1_P118 :=[[-111.1320078125,50.5559765625,0.53896728515625],[-7.8362214742082E-08,0.00132363335464177,5.92023053405581E-05,0.999999122244526],[0,0,0,0],[8.999999E+09,8.999999E+09,8.999999E+09,8.999999E+09,8.999999E+09,8.999999E+09]];
	LOCAL CONST Robtarget Tr_meulage_motif_1_P119 :=[[-111.571296875,51.45425390625,0.528108276367187],[-7.8362214742082E-08,0.00132363335464177,5.92023053405581E-05,0.999999122244526],[0,0,0,0],[8.999999E+09,8.999999E+09,8.999999E+09,8.999999E+09,8.999999E+09,8.999999E+09]];
	LOCAL CONST Robtarget Tr_meulage_motif_1_P120 :=[[-112.01059375,52.35253515625,0.517249328613281],[-7.8362214742082E-08,0.00132363335464177,5.92023053405581E-05,0.999999122244526],[0,0,0,0],[8.999999E+09,8.999999E+09,8.999999E+09,8.999999E+09,8.999999E+09,8.999999E+09]];
	LOCAL CONST Robtarget Tr_meulage_motif_1_P121 :=[[-112.4498828125,53.2508125,0.506390350341797],[-7.8362214742082E-08,0.00132363335464177,5.92023053405581E-05,0.999999122244526],[0,0,0,0],[8.999999E+09,8.999999E+09,8.999999E+09,8.999999E+09,8.999999E+09,8.999999E+09]];
	LOCAL CONST Robtarget Tr_meulage_motif_1_P122 :=[[-112.889171875,54.14908984375,0.495531341552734],[-7.8362214742082E-08,0.00132363335464177,5.92023053405581E-05,0.999999122244526],[0,0,0,0],[8.999999E+09,8.999999E+09,8.999999E+09,8.999999E+09,8.999999E+09,8.999999E+09]];
	LOCAL CONST Robtarget Tr_meulage_motif_1_P123 :=[[-113.32846875,55.0473671875,0.48467236328125],[-7.8362214742082E-08,0.00132363335464177,5.92023053405581E-05,0.999999122244526],[0,0,0,0],[8.999999E+09,8.999999E+09,8.999999E+09,8.999999E+09,8.999999E+09,8.999999E+09]];
	LOCAL CONST Robtarget Tr_meulage_motif_1_degg1 :=[[-113.354941393764,55.046183140358,-9.51529252651534],[-7.8362214742082E-08,0.00132363335464177,5.92023053405581E-05,0.999999122244526],[0,0,0,0],[8.999999E+09,8.999999E+09,8.999999E+09,8.999999E+09,8.999999E+09,8.999999E+09]];
	LOCAL CONST Robtarget Tr_meulage_motif_1_degg2 :=[[-113.85792162527,55.0236862446607,-199.514625432651],[-7.8362214742082E-08,0.00132363335464177,5.92023053405581E-05,0.999999122244526],[0,0,0,0],[8.999999E+09,8.999999E+09,8.999999E+09,8.999999E+09,8.999999E+09,8.999999E+09]];
	LOCAL CONST Robtarget Tr_meulage_motif_2_App1 :=[[240.648638261863,280.296146311066,26.5149057989462],[0.113971115605648,-0.110452064120549,-0.687112631333649,0.7090043428646],[0,0,0,0],[8.999999E+09,8.999999E+09,8.999999E+09,8.999999E+09,8.999999E+09,8.999999E+09]];
	LOCAL CONST Robtarget Tr_meulage_motif_2_App2 :=[[181.132283475593,99.9566983311783,32.4720036883848],[0.113971115605648,-0.110452064120549,-0.687112631333649,0.7090043428646],[0,0,0,0],[8.999999E+09,8.999999E+09,8.999999E+09,8.999999E+09,8.999999E+09,8.999999E+09]];
	LOCAL CONST Robtarget Tr_meulage_motif_2_P0 :=[[177.99984375,90.4651484375,32.78553515625],[0.113971115605648,-0.110452064120549,-0.687112631333649,0.7090043428646],[0,0,0,0],[8.999999E+09,8.999999E+09,8.999999E+09,8.999999E+09,8.999999E+09,8.999999E+09]];
	LOCAL CONST Robtarget Tr_meulage_motif_2_P1 :=[[177.046765625,90.767875,32.78553515625],[0.113971115605648,-0.110452064120549,-0.687112631333649,0.7090043428646],[0,0,0,0],[8.999999E+09,8.999999E+09,8.999999E+09,8.999999E+09,8.999999E+09,8.999999E+09]];
	LOCAL CONST Robtarget Tr_meulage_motif_2_P2 :=[[176.0936875,91.07059375,32.78553515625],[0.113971115605648,-0.110452064120549,-0.687112631333649,0.7090043428646],[0,0,0,0],[8.999999E+09,8.999999E+09,8.999999E+09,8.999999E+09,8.999999E+09,8.999999E+09]];
	LOCAL CONST Robtarget Tr_meulage_motif_2_P3 :=[[175.140609375,91.3733203125,32.78553515625],[0.113971115605648,-0.110452064120549,-0.687112631333649,0.7090043428646],[0,0,0,0],[8.999999E+09,8.999999E+09,8.999999E+09,8.999999E+09,8.999999E+09,8.999999E+09]];
	LOCAL CONST Robtarget Tr_meulage_motif_2_P4 :=[[174.18753125,91.6760390625,32.78553515625],[0.113971115605648,-0.110452064120549,-0.687112631333649,0.7090043428646],[0,0,0,0],[8.999999E+09,8.999999E+09,8.999999E+09,8.999999E+09,8.999999E+09,8.999999E+09]];
	LOCAL CONST Robtarget Tr_meulage_motif_2_P5 :=[[173.234453125,91.9787578125,32.78553515625],[0.113971115605648,-0.110452064120549,-0.687112631333649,0.7090043428646],[0,0,0,0],[8.999999E+09,8.999999E+09,8.999999E+09,8.999999E+09,8.999999E+09,8.999999E+09]];
	LOCAL CONST Robtarget Tr_meulage_motif_2_P6 :=[[172.281375,92.281484375,32.78553515625],[0.113971115605648,-0.110452064120549,-0.687112631333649,0.7090043428646],[0,0,0,0],[8.999999E+09,8.999999E+09,8.999999E+09,8.999999E+09,8.999999E+09,8.999999E+09]];
	LOCAL CONST Robtarget Tr_meulage_motif_2_P7 :=[[171.328296875,92.584203125,32.78553515625],[0.113971115605648,-0.110452064120549,-0.687112631333649,0.7090043428646],[0,0,0,0],[8.999999E+09,8.999999E+09,8.999999E+09,8.999999E+09,8.999999E+09,8.999999E+09]];
	LOCAL CONST Robtarget Tr_meulage_motif_2_P8 :=[[170.37521875,92.8869296875,32.78553515625],[0.113971115605648,-0.110452064120549,-0.687112631333649,0.7090043428646],[0,0,0,0],[8.999999E+09,8.999999E+09,8.999999E+09,8.999999E+09,8.999999E+09,8.999999E+09]];
	LOCAL CONST Robtarget Tr_meulage_motif_2_P9 :=[[169.422140625,93.1896484375,32.78553515625],[0.113971115605648,-0.110452064120549,-0.687112631333649,0.7090043428646],[0,0,0,0],[8.999999E+09,8.999999E+09,8.999999E+09,8.999999E+09,8.999999E+09,8.999999E+09]];
	LOCAL CONST Robtarget Tr_meulage_motif_2_P10 :=[[168.4690625,93.492375,32.78553515625],[0.113971115605648,-0.110452064120549,-0.687112631333649,0.7090043428646],[0,0,0,0],[8.999999E+09,8.999999E+09,8.999999E+09,8.999999E+09,8.999999E+09,8.999999E+09]];
	LOCAL CONST Robtarget Tr_meulage_motif_2_P11 :=[[167.515984375,93.79509375,32.78553515625],[0.113971115605648,-0.110452064120549,-0.687112631333649,0.7090043428646],[0,0,0,0],[8.999999E+09,8.999999E+09,8.999999E+09,8.999999E+09,8.999999E+09,8.999999E+09]];
	LOCAL CONST Robtarget Tr_meulage_motif_2_P12 :=[[166.56290625,94.0978203125,32.78553515625],[0.113971115605648,-0.110452064120549,-0.687112631333649,0.7090043428646],[0,0,0,0],[8.999999E+09,8.999999E+09,8.999999E+09,8.999999E+09,8.999999E+09,8.999999E+09]];
	LOCAL CONST Robtarget Tr_meulage_motif_2_P13 :=[[165.609828125,94.4005390625,32.78553515625],[0.113971115605648,-0.110452064120549,-0.687112631333649,0.7090043428646],[0,0,0,0],[8.999999E+09,8.999999E+09,8.999999E+09,8.999999E+09,8.999999E+09,8.999999E+09]];
	LOCAL CONST Robtarget Tr_meulage_motif_2_P14 :=[[164.65675,94.703265625,32.78553515625],[0.113971115605648,-0.110452064120549,-0.687112631333649,0.7090043428646],[0,0,0,0],[8.999999E+09,8.999999E+09,8.999999E+09,8.999999E+09,8.999999E+09,8.999999E+09]];
	LOCAL CONST Robtarget Tr_meulage_motif_2_P15 :=[[163.703671875,95.005984375,32.78553515625],[0.113971115605648,-0.110452064120549,-0.687112631333649,0.7090043428646],[0,0,0,0],[8.999999E+09,8.999999E+09,8.999999E+09,8.999999E+09,8.999999E+09,8.999999E+09]];
	LOCAL CONST Robtarget Tr_meulage_motif_2_P16 :=[[162.75059375,95.3087109375,32.78553515625],[0.113971115605648,-0.110452064120549,-0.687112631333649,0.7090043428646],[0,0,0,0],[8.999999E+09,8.999999E+09,8.999999E+09,8.999999E+09,8.999999E+09,8.999999E+09]];
	LOCAL CONST Robtarget Tr_meulage_motif_2_P17 :=[[161.797515625,95.6114296875,32.78553515625],[0.113971115605648,-0.110452064120549,-0.687112631333649,0.7090043428646],[0,0,0,0],[8.999999E+09,8.999999E+09,8.999999E+09,8.999999E+09,8.999999E+09,8.999999E+09]];
	LOCAL CONST Robtarget Tr_meulage_motif_2_P18 :=[[160.8444375,95.9141484375,32.78553515625],[0.113971115605648,-0.110452064120549,-0.687112631333649,0.7090043428646],[0,0,0,0],[8.999999E+09,8.999999E+09,8.999999E+09,8.999999E+09,8.999999E+09,8.999999E+09]];
	LOCAL CONST Robtarget Tr_meulage_motif_2_P19 :=[[159.898421875,96.2145625,32.674943359375],[0.113971115605648,-0.110452064120549,-0.687112631333649,0.7090043428646],[0,0,0,0],[8.999999E+09,8.999999E+09,8.999999E+09,8.999999E+09,8.999999E+09,8.999999E+09]];
	LOCAL CONST Robtarget Tr_meulage_motif_2_P20 :=[[158.996296875,96.50096875,32.463755859375],[0.113971115605648,-0.110452064120549,-0.687112631333649,0.7090043428646],[0,0,0,0],[8.999999E+09,8.999999E+09,8.999999E+09,8.999999E+09,8.999999E+09,8.999999E+09]];
	LOCAL CONST Robtarget Tr_meulage_motif_2_P21 :=[[158.18353125,96.7589453125,32.191912109375],[0.113971115605648,-0.110452064120549,-0.687112631333649,0.7090043428646],[0,0,0,0],[8.999999E+09,8.999999E+09,8.999999E+09,8.999999E+09,8.999999E+09,8.999999E+09]];
	LOCAL CONST Robtarget Tr_meulage_motif_2_P22 :=[[157.468734375,96.9858125,31.915974609375],[0.113971115605648,-0.110452064120549,-0.687112631333649,0.7090043428646],[0,0,0,0],[8.999999E+09,8.999999E+09,8.999999E+09,8.999999E+09,8.999999E+09,8.999999E+09]];
	LOCAL CONST Robtarget Tr_meulage_motif_2_P23 :=[[156.41921875,97.31878125,31.299849609375],[0.113971115605648,-0.110452064120549,-0.687112631333649,0.7090043428646],[0,0,0,0],[8.999999E+09,8.999999E+09,8.999999E+09,8.999999E+09,8.999999E+09,8.999999E+09]];
	LOCAL CONST Robtarget Tr_meulage_motif_2_P24 :=[[155.443234375,97.6282421875,30.452193359375],[0.113971115605648,-0.110452064120549,-0.687112631333649,0.7090043428646],[0,0,0,0],[8.999999E+09,8.999999E+09,8.999999E+09,8.999999E+09,8.999999E+09,8.999999E+09]];
	LOCAL CONST Robtarget Tr_meulage_motif_2_P25 :=[[154.635171875,97.884265625,29.4283203125],[0.113971115605648,-0.110452064120549,-0.687112631333649,0.7090043428646],[0,0,0,0],[8.999999E+09,8.999999E+09,8.999999E+09,8.999999E+09,8.999999E+09,8.999999E+09]];
	LOCAL CONST Robtarget Tr_meulage_motif_2_P26 :=[[154.16971875,98.03140625,28.3121328125],[0.113971115605648,-0.110452064120549,-0.687112631333649,0.7090043428646],[0,0,0,0],[8.999999E+09,8.999999E+09,8.999999E+09,8.999999E+09,8.999999E+09,8.999999E+09]];
	LOCAL CONST Robtarget Tr_meulage_motif_2_P27 :=[[154.143796875,98.039203125,27.6161640625],[0.113971115605648,-0.110452064120549,-0.687112631333649,0.7090043428646],[0,0,0,0],[8.999999E+09,8.999999E+09,8.999999E+09,8.999999E+09,8.999999E+09,8.999999E+09]];
	LOCAL CONST Robtarget Tr_meulage_motif_2_P28 :=[[154.143671875,98.0388203125,26.9549140625],[0.113971115605648,-0.110452064120549,-0.687112631333649,0.7090043428646],[0,0,0,0],[8.999999E+09,8.999999E+09,8.999999E+09,8.999999E+09,8.999999E+09,8.999999E+09]];
	LOCAL CONST Robtarget Tr_meulage_motif_2_P29 :=[[154.195859375,98.0218359375,26.2938203125],[0.113971115605648,-0.110452064120549,-0.687112631333649,0.7090043428646],[0,0,0,0],[8.999999E+09,8.999999E+09,8.999999E+09,8.999999E+09,8.999999E+09,8.999999E+09]];
	LOCAL CONST Robtarget Tr_meulage_motif_2_P30 :=[[154.6705,97.8703828125,25.1920703125],[0.113971115605648,-0.110452064120549,-0.687112631333649,0.7090043428646],[0,0,0,0],[8.999999E+09,8.999999E+09,8.999999E+09,8.999999E+09,8.999999E+09,8.999999E+09]];
	LOCAL CONST Robtarget Tr_meulage_motif_2_P31 :=[[155.48675,97.6104921875,24.1854453125],[0.113971115605648,-0.110452064120549,-0.687112631333649,0.7090043428646],[0,0,0,0],[8.999999E+09,8.999999E+09,8.999999E+09,8.999999E+09,8.999999E+09,8.999999E+09]];
	LOCAL CONST Robtarget Tr_meulage_motif_2_P32 :=[[156.461984375,97.3002109375,23.3565703125],[0.113971115605648,-0.110452064120549,-0.687112631333649,0.7090043428646],[0,0,0,0],[8.999999E+09,8.999999E+09,8.999999E+09,8.999999E+09,8.999999E+09,8.999999E+09]];
	LOCAL CONST Robtarget Tr_meulage_motif_2_P33 :=[[157.116765625,97.091984375,22.9608203125],[0.113971115605648,-0.110452064120549,-0.687112631333649,0.7090043428646],[0,0,0,0],[8.999999E+09,8.999999E+09,8.999999E+09,8.999999E+09,8.999999E+09,8.999999E+09]];
	LOCAL CONST Robtarget Tr_meulage_motif_2_P34 :=[[158.2205,96.741109375,22.4732890625],[0.113971115605648,-0.110452064120549,-0.687112631333649,0.7090043428646],[0,0,0,0],[8.999999E+09,8.999999E+09,8.999999E+09,8.999999E+09,8.999999E+09,8.999999E+09]];
	LOCAL CONST Robtarget Tr_meulage_motif_2_P35 :=[[159.025828125,96.4851484375,22.2091953125],[0.113971115605648,-0.110452064120549,-0.687112631333649,0.7090043428646],[0,0,0,0],[8.999999E+09,8.999999E+09,8.999999E+09,8.999999E+09,8.999999E+09,8.999999E+09]];
	LOCAL CONST Robtarget Tr_meulage_motif_2_P36 :=[[159.9140625,96.202890625,22.0047265625],[0.113971115605648,-0.110452064120549,-0.687112631333649,0.7090043428646],[0,0,0,0],[8.999999E+09,8.999999E+09,8.999999E+09,8.999999E+09,8.999999E+09,8.999999E+09]];
	LOCAL CONST Robtarget Tr_meulage_motif_2_P37 :=[[160.849546875,95.9056875,21.8961328125],[0.113971115605648,-0.110452064120549,-0.687112631333649,0.7090043428646],[0,0,0,0],[8.999999E+09,8.999999E+09,8.999999E+09,8.999999E+09,8.999999E+09,8.999999E+09]];
	LOCAL CONST Robtarget Tr_meulage_motif_2_P38 :=[[161.795515625,95.60515625,21.7855390625],[0.113971115605648,-0.110452064120549,-0.687112631333649,0.7090043428646],[0,0,0,0],[8.999999E+09,8.999999E+09,8.999999E+09,8.999999E+09,8.999999E+09,8.999999E+09]];
	LOCAL CONST Robtarget Tr_meulage_motif_2_P39 :=[[162.74859375,95.3024296875,21.7855390625],[0.113971115605648,-0.110452064120549,-0.687112631333649,0.7090043428646],[0,0,0,0],[8.999999E+09,8.999999E+09,8.999999E+09,8.999999E+09,8.999999E+09,8.999999E+09]];
	LOCAL CONST Robtarget Tr_meulage_motif_2_P40 :=[[163.701671875,94.9997109375,21.7855390625],[0.113971115605648,-0.110452064120549,-0.687112631333649,0.7090043428646],[0,0,0,0],[8.999999E+09,8.999999E+09,8.999999E+09,8.999999E+09,8.999999E+09,8.999999E+09]];
	LOCAL CONST Robtarget Tr_meulage_motif_2_P41 :=[[164.65475,94.696984375,21.7855390625],[0.113971115605648,-0.110452064120549,-0.687112631333649,0.7090043428646],[0,0,0,0],[8.999999E+09,8.999999E+09,8.999999E+09,8.999999E+09,8.999999E+09,8.999999E+09]];
	LOCAL CONST Robtarget Tr_meulage_motif_2_P42 :=[[165.607828125,94.394265625,21.7855390625],[0.113971115605648,-0.110452064120549,-0.687112631333649,0.7090043428646],[0,0,0,0],[8.999999E+09,8.999999E+09,8.999999E+09,8.999999E+09,8.999999E+09,8.999999E+09]];
	LOCAL CONST Robtarget Tr_meulage_motif_2_P43 :=[[166.56090625,94.0915390625,21.7855390625],[0.113971115605648,-0.110452064120549,-0.687112631333649,0.7090043428646],[0,0,0,0],[8.999999E+09,8.999999E+09,8.999999E+09,8.999999E+09,8.999999E+09,8.999999E+09]];
	LOCAL CONST Robtarget Tr_meulage_motif_2_P44 :=[[167.513984375,93.7888203125,21.7855390625],[0.113971115605648,-0.110452064120549,-0.687112631333649,0.7090043428646],[0,0,0,0],[8.999999E+09,8.999999E+09,8.999999E+09,8.999999E+09,8.999999E+09,8.999999E+09]];
	LOCAL CONST Robtarget Tr_meulage_motif_2_P45 :=[[168.4670625,93.4861015625,21.7855390625],[0.113971115605648,-0.110452064120549,-0.687112631333649,0.7090043428646],[0,0,0,0],[8.999999E+09,8.999999E+09,8.999999E+09,8.999999E+09,8.999999E+09,8.999999E+09]];
	LOCAL CONST Robtarget Tr_meulage_motif_2_P46 :=[[169.420140625,93.183375,21.7855390625],[0.113971115605648,-0.110452064120549,-0.687112631333649,0.7090043428646],[0,0,0,0],[8.999999E+09,8.999999E+09,8.999999E+09,8.999999E+09,8.999999E+09,8.999999E+09]];
	LOCAL CONST Robtarget Tr_meulage_motif_2_P47 :=[[170.37321875,92.88065625,21.7855390625],[0.113971115605648,-0.110452064120549,-0.687112631333649,0.7090043428646],[0,0,0,0],[8.999999E+09,8.999999E+09,8.999999E+09,8.999999E+09,8.999999E+09,8.999999E+09]];
	LOCAL CONST Robtarget Tr_meulage_motif_2_P48 :=[[171.326296875,92.5779296875,21.7855390625],[0.113971115605648,-0.110452064120549,-0.687112631333649,0.7090043428646],[0,0,0,0],[8.999999E+09,8.999999E+09,8.999999E+09,8.999999E+09,8.999999E+09,8.999999E+09]];
	LOCAL CONST Robtarget Tr_meulage_motif_2_P49 :=[[172.27228125,92.2773984375,21.674943359375],[0.113971115605648,-0.110452064120549,-0.687112631333649,0.7090043428646],[0,0,0,0],[8.999999E+09,8.999999E+09,8.999999E+09,8.999999E+09,8.999999E+09,8.999999E+09]];
	LOCAL CONST Robtarget Tr_meulage_motif_2_P50 :=[[173.174328125,91.99075,21.463755859375],[0.113971115605648,-0.110452064120549,-0.687112631333649,0.7090043428646],[0,0,0,0],[8.999999E+09,8.999999E+09,8.999999E+09,8.999999E+09,8.999999E+09,8.999999E+09]];
	LOCAL CONST Robtarget Tr_meulage_motif_2_P51 :=[[173.986984375,91.7324609375,21.191912109375],[0.113971115605648,-0.110452064120549,-0.687112631333649,0.7090043428646],[0,0,0,0],[8.999999E+09,8.999999E+09,8.999999E+09,8.999999E+09,8.999999E+09,8.999999E+09]];
	LOCAL CONST Robtarget Tr_meulage_motif_2_P52 :=[[174.665046875,91.5168984375,20.887755859375],[0.113971115605648,-0.110452064120549,-0.687112631333649,0.7090043428646],[0,0,0,0],[8.999999E+09,8.999999E+09,8.999999E+09,8.999999E+09,8.999999E+09,8.999999E+09]];
	LOCAL CONST Robtarget Tr_meulage_motif_2_P53 :=[[175.650859375,91.203359375,20.225224609375],[0.113971115605648,-0.110452064120549,-0.687112631333649,0.7090043428646],[0,0,0,0],[8.999999E+09,8.999999E+09,8.999999E+09,8.999999E+09,8.999999E+09,8.999999E+09]];
	LOCAL CONST Robtarget Tr_meulage_motif_2_P54 :=[[176.5103125,90.9298125,19.3232890625],[0.113971115605648,-0.110452064120549,-0.687112631333649,0.7090043428646],[0,0,0,0],[8.999999E+09,8.999999E+09,8.999999E+09,8.999999E+09,8.999999E+09,8.999999E+09]];
	LOCAL CONST Robtarget Tr_meulage_motif_2_P55 :=[[177.019984375,90.767265625,18.2772578125],[0.113971115605648,-0.110452064120549,-0.687112631333649,0.7090043428646],[0,0,0,0],[8.999999E+09,8.999999E+09,8.999999E+09,8.999999E+09,8.999999E+09,8.999999E+09]];
	LOCAL CONST Robtarget Tr_meulage_motif_2_P56 :=[[177.19596875,90.7109375,17.5840390625],[0.113971115605648,-0.110452064120549,-0.687112631333649,0.7090043428646],[0,0,0,0],[8.999999E+09,8.999999E+09,8.999999E+09,8.999999E+09,8.999999E+09,8.999999E+09]];
	LOCAL CONST Robtarget Tr_meulage_motif_2_P57 :=[[177.2566875,90.691171875,16.8140390625],[0.113971115605648,-0.110452064120549,-0.687112631333649,0.7090043428646],[0,0,0,0],[8.999999E+09,8.999999E+09,8.999999E+09,8.999999E+09,8.999999E+09,8.999999E+09]];
	LOCAL CONST Robtarget Tr_meulage_motif_2_P58 :=[[177.19275,90.7109921875,16.0441640625],[0.113971115605648,-0.110452064120549,-0.687112631333649,0.7090043428646],[0,0,0,0],[8.999999E+09,8.999999E+09,8.999999E+09,8.999999E+09,8.999999E+09,8.999999E+09]];
	LOCAL CONST Robtarget Tr_meulage_motif_2_P59 :=[[176.792640625,90.8373828125,14.9359140625],[0.113971115605648,-0.110452064120549,-0.687112631333649,0.7090043428646],[0,0,0,0],[8.999999E+09,8.999999E+09,8.999999E+09,8.999999E+09,8.999999E+09,8.999999E+09]];
	LOCAL CONST Robtarget Tr_meulage_motif_2_P60 :=[[176.39765625,90.96246875,14.3502265625],[0.113971115605648,-0.110452064120549,-0.687112631333649,0.7090043428646],[0,0,0,0],[8.999999E+09,8.999999E+09,8.999999E+09,8.999999E+09,8.999999E+09,8.999999E+09]];
	LOCAL CONST Robtarget Tr_meulage_motif_2_P61 :=[[175.552,91.230515625,13.4631015625],[0.113971115605648,-0.110452064120549,-0.687112631333649,0.7090043428646],[0,0,0,0],[8.999999E+09,8.999999E+09,8.999999E+09,8.999999E+09,8.999999E+09,8.999999E+09]];
	LOCAL CONST Robtarget Tr_meulage_motif_2_P62 :=[[174.99371875,91.407578125,13.0487890625],[0.113971115605648,-0.110452064120549,-0.687112631333649,0.7090043428646],[0,0,0,0],[8.999999E+09,8.999999E+09,8.999999E+09,8.999999E+09,8.999999E+09,8.999999E+09]];
	LOCAL CONST Robtarget Tr_meulage_motif_2_P63 :=[[173.928171875,91.7456875,12.5046953125],[0.113971115605648,-0.110452064120549,-0.687112631333649,0.7090043428646],[0,0,0,0],[8.999999E+09,8.999999E+09,8.999999E+09,8.999999E+09,8.999999E+09,8.999999E+09]];
	LOCAL CONST Robtarget Tr_meulage_motif_2_P64 :=[[173.14125,91.9954453125,12.2091962890625],[0.113971115605648,-0.110452064120549,-0.687112631333649,0.7090043428646],[0,0,0,0],[8.999999E+09,8.999999E+09,8.999999E+09,8.999999E+09,8.999999E+09,8.999999E+09]];
	LOCAL CONST Robtarget Tr_meulage_motif_2_P65 :=[[172.252953125,92.2774609375,12.0047275390625],[0.113971115605648,-0.110452064120549,-0.687112631333649,0.7090043428646],[0,0,0,0],[8.999999E+09,8.999999E+09,8.999999E+09,8.999999E+09,8.999999E+09,8.999999E+09]];
	LOCAL CONST Robtarget Tr_meulage_motif_2_P66 :=[[171.317421875,92.5745390625,11.8961337890625],[0.113971115605648,-0.110452064120549,-0.687112631333649,0.7090043428646],[0,0,0,0],[8.999999E+09,8.999999E+09,8.999999E+09,8.999999E+09,8.999999E+09,8.999999E+09]];
	LOCAL CONST Robtarget Tr_meulage_motif_2_P67 :=[[170.37140625,92.8749453125,11.7855400390625],[0.113971115605648,-0.110452064120549,-0.687112631333649,0.7090043428646],[0,0,0,0],[8.999999E+09,8.999999E+09,8.999999E+09,8.999999E+09,8.999999E+09,8.999999E+09]];
	LOCAL CONST Robtarget Tr_meulage_motif_2_P68 :=[[169.418328125,93.177671875,11.7855400390625],[0.113971115605648,-0.110452064120549,-0.687112631333649,0.7090043428646],[0,0,0,0],[8.999999E+09,8.999999E+09,8.999999E+09,8.999999E+09,8.999999E+09,8.999999E+09]];
	LOCAL CONST Robtarget Tr_meulage_motif_2_P69 :=[[168.46525,93.480390625,11.7855400390625],[0.113971115605648,-0.110452064120549,-0.687112631333649,0.7090043428646],[0,0,0,0],[8.999999E+09,8.999999E+09,8.999999E+09,8.999999E+09,8.999999E+09,8.999999E+09]];
	LOCAL CONST Robtarget Tr_meulage_motif_2_P70 :=[[167.512171875,93.7831171875,11.7855400390625],[0.113971115605648,-0.110452064120549,-0.687112631333649,0.7090043428646],[0,0,0,0],[8.999999E+09,8.999999E+09,8.999999E+09,8.999999E+09,8.999999E+09,8.999999E+09]];
	LOCAL CONST Robtarget Tr_meulage_motif_2_P71 :=[[166.55909375,94.0858359375,11.7855400390625],[0.113971115605648,-0.110452064120549,-0.687112631333649,0.7090043428646],[0,0,0,0],[8.999999E+09,8.999999E+09,8.999999E+09,8.999999E+09,8.999999E+09,8.999999E+09]];
	LOCAL CONST Robtarget Tr_meulage_motif_2_P72 :=[[165.606015625,94.3885625,11.7855400390625],[0.113971115605648,-0.110452064120549,-0.687112631333649,0.7090043428646],[0,0,0,0],[8.999999E+09,8.999999E+09,8.999999E+09,8.999999E+09,8.999999E+09,8.999999E+09]];
	LOCAL CONST Robtarget Tr_meulage_motif_2_P73 :=[[164.6529375,94.69128125,11.7855400390625],[0.113971115605648,-0.110452064120549,-0.687112631333649,0.7090043428646],[0,0,0,0],[8.999999E+09,8.999999E+09,8.999999E+09,8.999999E+09,8.999999E+09,8.999999E+09]];
	LOCAL CONST Robtarget Tr_meulage_motif_2_P74 :=[[163.699859375,94.9940078125,11.785541015625],[0.113971115605648,-0.110452064120549,-0.687112631333649,0.7090043428646],[0,0,0,0],[8.999999E+09,8.999999E+09,8.999999E+09,8.999999E+09,8.999999E+09,8.999999E+09]];
	LOCAL CONST Robtarget Tr_meulage_motif_2_P75 :=[[162.74678125,95.2967265625,11.785541015625],[0.113971115605648,-0.110452064120549,-0.687112631333649,0.7090043428646],[0,0,0,0],[8.999999E+09,8.999999E+09,8.999999E+09,8.999999E+09,8.999999E+09,8.999999E+09]];
	LOCAL CONST Robtarget Tr_meulage_motif_2_P76 :=[[161.793703125,95.599453125,11.785541015625],[0.113971115605648,-0.110452064120549,-0.687112631333649,0.7090043428646],[0,0,0,0],[8.999999E+09,8.999999E+09,8.999999E+09,8.999999E+09,8.999999E+09,8.999999E+09]];
	LOCAL CONST Robtarget Tr_meulage_motif_2_P77 :=[[160.840625,95.902171875,11.785541015625],[0.113971115605648,-0.110452064120549,-0.687112631333649,0.7090043428646],[0,0,0,0],[8.999999E+09,8.999999E+09,8.999999E+09,8.999999E+09,8.999999E+09,8.999999E+09]];
	LOCAL CONST Robtarget Tr_meulage_motif_2_P78 :=[[159.894609375,96.202578125,11.674947265625],[0.113971115605648,-0.110452064120549,-0.687112631333649,0.7090043428646],[0,0,0,0],[8.999999E+09,8.999999E+09,8.999999E+09,8.999999E+09,8.999999E+09,8.999999E+09]];
	LOCAL CONST Robtarget Tr_meulage_motif_2_P79 :=[[158.992484375,96.488984375,11.463759765625],[0.113971115605648,-0.110452064120549,-0.687112631333649,0.7090043428646],[0,0,0,0],[8.999999E+09,8.999999E+09,8.999999E+09,8.999999E+09,8.999999E+09,8.999999E+09]];
	LOCAL CONST Robtarget Tr_meulage_motif_2_P80 :=[[158.179734375,96.74696875,11.191916015625],[0.113971115605648,-0.110452064120549,-0.687112631333649,0.7090043428646],[0,0,0,0],[8.999999E+09,8.999999E+09,8.999999E+09,8.999999E+09,8.999999E+09,8.999999E+09]];
	LOCAL CONST Robtarget Tr_meulage_motif_2_P81 :=[[157.4649375,96.9738359375,10.915978515625],[0.113971115605648,-0.110452064120549,-0.687112631333649,0.7090043428646],[0,0,0,0],[8.999999E+09,8.999999E+09,8.999999E+09,8.999999E+09,8.999999E+09,8.999999E+09]];
	LOCAL CONST Robtarget Tr_meulage_motif_2_P82 :=[[156.415421875,97.306796875,10.299853515625],[0.113971115605648,-0.110452064120549,-0.687112631333649,0.7090043428646],[0,0,0,0],[8.999999E+09,8.999999E+09,8.999999E+09,8.999999E+09,8.999999E+09,8.999999E+09]];
	LOCAL CONST Robtarget Tr_meulage_motif_2_P83 :=[[155.503421875,97.59590625,9.4058857421875],[0.113971115605648,-0.110452064120549,-0.687112631333649,0.7090043428646],[0,0,0,0],[8.999999E+09,8.999999E+09,8.999999E+09,8.999999E+09,8.999999E+09,8.999999E+09]];
	LOCAL CONST Robtarget Tr_meulage_motif_2_P84 :=[[154.9226875,97.7796875,8.3198857421875],[0.113971115605648,-0.110452064120549,-0.687112631333649,0.7090043428646],[0,0,0,0],[8.999999E+09,8.999999E+09,8.999999E+09,8.999999E+09,8.999999E+09,8.999999E+09]];
	LOCAL CONST Robtarget Tr_meulage_motif_2_P85 :=[[154.761140625,97.830375,7.3355107421875],[0.113971115605648,-0.110452064120549,-0.687112631333649,0.7090043428646],[0,0,0,0],[8.999999E+09,8.999999E+09,8.999999E+09,8.999999E+09,8.999999E+09,8.999999E+09]];
	LOCAL CONST Robtarget Tr_meulage_motif_2_P86 :=[[154.88640625,97.7904609375,7.1308544921875],[0.113971115605648,-0.110452064120549,-0.687112631333649,0.7090043428646],[0,0,0,0],[8.999999E+09,8.999999E+09,8.999999E+09,8.999999E+09,8.999999E+09,8.999999E+09]];
	LOCAL CONST Robtarget Tr_meulage_motif_2_P87 :=[[155.003859375,97.752703125,6.40444873046875],[0.113971115605648,-0.110452064120549,-0.687112631333649,0.7090043428646],[0,0,0,0],[8.999999E+09,8.999999E+09,8.999999E+09,8.999999E+09,8.999999E+09,8.999999E+09]];
	LOCAL CONST Robtarget Tr_meulage_motif_2_P88 :=[[155.65559375,97.5451015625,5.46754248046875],[0.113971115605648,-0.110452064120549,-0.687112631333649,0.7090043428646],[0,0,0,0],[8.999999E+09,8.999999E+09,8.999999E+09,8.999999E+09,8.999999E+09,8.999999E+09]];
	LOCAL CONST Robtarget Tr_meulage_motif_2_P89 :=[[156.18696875,97.37603125,5.00372998046875],[0.113971115605648,-0.110452064120549,-0.687112631333649,0.7090043428646],[0,0,0,0],[8.999999E+09,8.999999E+09,8.999999E+09,8.999999E+09,8.999999E+09,8.999999E+09]];
	LOCAL CONST Robtarget Tr_meulage_motif_2_P90 :=[[157.26415625,97.0335625,4.47329248046875],[0.113971115605648,-0.110452064120549,-0.687112631333649,0.7090043428646],[0,0,0,0],[8.999999E+09,8.999999E+09,8.999999E+09,8.999999E+09,8.999999E+09,8.999999E+09]];
	LOCAL CONST Robtarget Tr_meulage_motif_2_P91 :=[[158.069484375,96.7776015625,4.20919873046875],[0.113971115605648,-0.110452064120549,-0.687112631333649,0.7090043428646],[0,0,0,0],[8.999999E+09,8.999999E+09,8.999999E+09,8.999999E+09,8.999999E+09,8.999999E+09]];
	LOCAL CONST Robtarget Tr_meulage_motif_2_P92 :=[[158.95771875,96.49534375,4.00472998046875],[0.113971115605648,-0.110452064120549,-0.687112631333649,0.7090043428646],[0,0,0,0],[8.999999E+09,8.999999E+09,8.999999E+09,8.999999E+09,8.999999E+09,8.999999E+09]];
	LOCAL CONST Robtarget Tr_meulage_motif_2_P93 :=[[159.893203125,96.198140625,3.89613598632813],[0.113971115605648,-0.110452064120549,-0.687112631333649,0.7090043428646],[0,0,0,0],[8.999999E+09,8.999999E+09,8.999999E+09,8.999999E+09,8.999999E+09,8.999999E+09]];
	LOCAL CONST Robtarget Tr_meulage_motif_2_P94 :=[[160.839171875,95.897609375,3.78554223632813],[0.113971115605648,-0.110452064120549,-0.687112631333649,0.7090043428646],[0,0,0,0],[8.999999E+09,8.999999E+09,8.999999E+09,8.999999E+09,8.999999E+09,8.999999E+09]];
	LOCAL CONST Robtarget Tr_meulage_motif_2_P95 :=[[161.79225,95.5948828125,3.78554223632813],[0.113971115605648,-0.110452064120549,-0.687112631333649,0.7090043428646],[0,0,0,0],[8.999999E+09,8.999999E+09,8.999999E+09,8.999999E+09,8.999999E+09,8.999999E+09]];
	LOCAL CONST Robtarget Tr_meulage_motif_2_P96 :=[[162.745328125,95.2921640625,3.7855419921875],[0.113971115605648,-0.110452064120549,-0.687112631333649,0.7090043428646],[0,0,0,0],[8.999999E+09,8.999999E+09,8.999999E+09,8.999999E+09,8.999999E+09,8.999999E+09]];
	LOCAL CONST Robtarget Tr_meulage_motif_2_P97 :=[[163.69840625,94.9894453125,3.7855419921875],[0.113971115605648,-0.110452064120549,-0.687112631333649,0.7090043428646],[0,0,0,0],[8.999999E+09,8.999999E+09,8.999999E+09,8.999999E+09,8.999999E+09,8.999999E+09]];
	LOCAL CONST Robtarget Tr_meulage_motif_2_P98 :=[[164.651484375,94.68671875,3.7855419921875],[0.113971115605648,-0.110452064120549,-0.687112631333649,0.7090043428646],[0,0,0,0],[8.999999E+09,8.999999E+09,8.999999E+09,8.999999E+09,8.999999E+09,8.999999E+09]];
	LOCAL CONST Robtarget Tr_meulage_motif_2_P99 :=[[165.6045625,94.384,3.78554174804687],[0.113971115605648,-0.110452064120549,-0.687112631333649,0.7090043428646],[0,0,0,0],[8.999999E+09,8.999999E+09,8.999999E+09,8.999999E+09,8.999999E+09,8.999999E+09]];
	LOCAL CONST Robtarget Tr_meulage_motif_2_P100 :=[[166.557640625,94.0812734375,3.78554174804687],[0.113971115605648,-0.110452064120549,-0.687112631333649,0.7090043428646],[0,0,0,0],[8.999999E+09,8.999999E+09,8.999999E+09,8.999999E+09,8.999999E+09,8.999999E+09]];
	LOCAL CONST Robtarget Tr_meulage_motif_2_P101 :=[[167.51071875,93.7785546875,3.78554174804687],[0.113971115605648,-0.110452064120549,-0.687112631333649,0.7090043428646],[0,0,0,0],[8.999999E+09,8.999999E+09,8.999999E+09,8.999999E+09,8.999999E+09,8.999999E+09]];
	LOCAL CONST Robtarget Tr_meulage_motif_2_P102 :=[[168.4638125,93.475828125,3.78554150390625],[0.113971115605648,-0.110452064120549,-0.687112631333649,0.7090043428646],[0,0,0,0],[8.999999E+09,8.999999E+09,8.999999E+09,8.999999E+09,8.999999E+09,8.999999E+09]];
	LOCAL CONST Robtarget Tr_meulage_motif_2_P103 :=[[169.416890625,93.173109375,3.78554150390625],[0.113971115605648,-0.110452064120549,-0.687112631333649,0.7090043428646],[0,0,0,0],[8.999999E+09,8.999999E+09,8.999999E+09,8.999999E+09,8.999999E+09,8.999999E+09]];
	LOCAL CONST Robtarget Tr_meulage_motif_2_P104 :=[[170.36996875,92.8703828125,3.78554150390625],[0.113971115605648,-0.110452064120549,-0.687112631333649,0.7090043428646],[0,0,0,0],[8.999999E+09,8.999999E+09,8.999999E+09,8.999999E+09,8.999999E+09,8.999999E+09]];
	LOCAL CONST Robtarget Tr_meulage_motif_2_P105 :=[[171.323046875,92.5676640625,3.78554125976563],[0.113971115605648,-0.110452064120549,-0.687112631333649,0.7090043428646],[0,0,0,0],[8.999999E+09,8.999999E+09,8.999999E+09,8.999999E+09,8.999999E+09,8.999999E+09]];
	LOCAL CONST Robtarget Tr_meulage_motif_2_P106 :=[[172.276125,92.2649375,3.78554125976563],[0.113971115605648,-0.110452064120549,-0.687112631333649,0.7090043428646],[0,0,0,0],[8.999999E+09,8.999999E+09,8.999999E+09,8.999999E+09,8.999999E+09,8.999999E+09]];
	LOCAL CONST Robtarget Tr_meulage_motif_2_P107 :=[[173.229203125,91.96221875,3.78554125976563],[0.113971115605648,-0.110452064120549,-0.687112631333649,0.7090043428646],[0,0,0,0],[8.999999E+09,8.999999E+09,8.999999E+09,8.999999E+09,8.999999E+09,8.999999E+09]];
	LOCAL CONST Robtarget Tr_meulage_motif_2_P108 :=[[174.18228125,91.6594921875,3.785541015625],[0.113971115605648,-0.110452064120549,-0.687112631333649,0.7090043428646],[0,0,0,0],[8.999999E+09,8.999999E+09,8.999999E+09,8.999999E+09,8.999999E+09,8.999999E+09]];
	LOCAL CONST Robtarget Tr_meulage_motif_2_P109 :=[[175.135359375,91.3567734375,3.785541015625],[0.113971115605648,-0.110452064120549,-0.687112631333649,0.7090043428646],[0,0,0,0],[8.999999E+09,8.999999E+09,8.999999E+09,8.999999E+09,8.999999E+09,8.999999E+09]];
	LOCAL CONST Robtarget Tr_meulage_motif_2_P110 :=[[176.0884375,91.0540546875,3.785541015625],[0.113971115605648,-0.110452064120549,-0.687112631333649,0.7090043428646],[0,0,0,0],[8.999999E+09,8.999999E+09,8.999999E+09,8.999999E+09,8.999999E+09,8.999999E+09]];
	LOCAL CONST Robtarget Tr_meulage_motif_2_P111 :=[[177.041515625,90.751328125,3.78554077148438],[0.113971115605648,-0.110452064120549,-0.687112631333649,0.7090043428646],[0,0,0,0],[8.999999E+09,8.999999E+09,8.999999E+09,8.999999E+09,8.999999E+09,8.999999E+09]];
	LOCAL CONST Robtarget Tr_meulage_motif_2_P112 :=[[177.99459375,90.448609375,3.78554077148438],[0.113971115605648,-0.110452064120549,-0.687112631333649,0.7090043428646],[0,0,0,0],[8.999999E+09,8.999999E+09,8.999999E+09,8.999999E+09,8.999999E+09,8.999999E+09]];
	LOCAL CONST Robtarget Tr_meulage_motif_2_P113 :=[[178.947671875,90.1458828125,3.78554077148438],[0.113971115605648,-0.110452064120549,-0.687112631333649,0.7090043428646],[0,0,0,0],[8.999999E+09,8.999999E+09,8.999999E+09,8.999999E+09,8.999999E+09,8.999999E+09]];
	LOCAL CONST Robtarget Tr_meulage_motif_2_P114 :=[[179.90075,89.8431640625,3.78554052734375],[0.113971115605648,-0.110452064120549,-0.687112631333649,0.7090043428646],[0,0,0,0],[8.999999E+09,8.999999E+09,8.999999E+09,8.999999E+09,8.999999E+09,8.999999E+09]];
	LOCAL CONST Robtarget Tr_meulage_motif_2_P115 :=[[180.853828125,89.5404375,3.78554052734375],[0.113971115605648,-0.110452064120549,-0.687112631333649,0.7090043428646],[0,0,0,0],[8.999999E+09,8.999999E+09,8.999999E+09,8.999999E+09,8.999999E+09,8.999999E+09]];
	LOCAL CONST Robtarget Tr_meulage_motif_2_degg1 :=[[183.986267850593,99.0319873936783,3.47200905947856],[0.113971115605648,-0.110452064120549,-0.687112631333649,0.7090043428646],[0,0,0,0],[8.999999E+09,8.999999E+09,8.999999E+09,8.999999E+09,8.999999E+09,8.999999E+09]];
	LOCAL CONST Robtarget Tr_meulage_motif_2_degg2 :=[[243.502622636863,279.371435373566,-2.48508882996003],[0.113971115605648,-0.110452064120549,-0.687112631333649,0.7090043428646],[0,0,0,0],[8.999999E+09,8.999999E+09,8.999999E+09,8.999999E+09,8.999999E+09,8.999999E+09]];
	LOCAL CONST Robtarget Tr_meulage_bavure_App1 :=[[-405.507038442101,-102.209165839799,19.2786571091216],[0.628166471153475,-0.638549991152604,0.316939349989573,-0.311785570137212],[0,0,0,0],[8.999999E+09,8.999999E+09,8.999999E+09,8.999999E+09,8.999999E+09,8.999999E+09]];
	LOCAL CONST Robtarget Tr_meulage_bavure_App2 :=[[-254.198126922105,12.66429405176,16.1639328554561],[0.628166471153475,-0.638549991152604,0.316939349989573,-0.311785570137212],[0,0,0,0],[8.999999E+09,8.999999E+09,8.999999E+09,8.999999E+09,8.999999E+09,8.999999E+09]];
	LOCAL CONST Robtarget Tr_meulage_bavure_P0 :=[[-246.2345,18.710265625,16],[0.628166471153475,-0.638549991152604,0.316939349989573,-0.311785570137212],[0,0,0,0],[8.999999E+09,8.999999E+09,8.999999E+09,8.999999E+09,8.999999E+09,8.999999E+09]];
	LOCAL CONST Robtarget Tr_meulage_bavure_P1 :=[[-246.761421875,19.243376953125,16],[0.627155815260354,-0.637868582745397,0.318734201882854,-0.313381178569485],[0,0,0,0],[8.999999E+09,8.999999E+09,8.999999E+09,8.999999E+09,8.999999E+09,8.999999E+09]];
	LOCAL CONST Robtarget Tr_meulage_bavure_P2 :=[[-247.493828125,20.18832421875,16],[0.624220819464608,-0.635920480041685,0.323865321610752,-0.317906849672117],[0,0,0,0],[8.999999E+09,8.999999E+09,8.999999E+09,8.999999E+09,8.999999E+09,8.999999E+09]];
	LOCAL CONST Robtarget Tr_meulage_bavure_P3 :=[[-249.746828125,22.29608203125,16],[0.619599333735136,-0.632908373297614,0.331740419121046,-0.324764454591534],[0,0,0,0],[8.999999E+09,8.999999E+09,8.999999E+09,8.999999E+09,8.999999E+09,8.999999E+09]];
	LOCAL CONST Robtarget Tr_meulage_bavure_P4 :=[[-251.414328125,24.411681640625,16],[0.613527654162665,-0.628998936438891,0.341774600518026,-0.333368081821198],[0,0,0,0],[8.999999E+09,8.999999E+09,8.999999E+09,8.999999E+09,8.999999E+09,8.999999E+09]];
	LOCAL CONST Robtarget Tr_meulage_bavure_P5 :=[[-252.126359375,25.32571484375,16],[0.606034920589616,-0.62416896057567,0.353766285775687,-0.343488280336171],[0,0,0,0],[8.999999E+09,8.999999E+09,8.999999E+09,8.999999E+09,8.999999E+09,8.999999E+09]];
	LOCAL CONST Robtarget Tr_meulage_bavure_P6 :=[[-252.223171875,25.484984375,16],[0.596860348338097,-0.618040011885802,0.368041435916354,-0.355428993947527],[0,0,0,0],[8.999999E+09,8.999999E+09,8.999999E+09,8.999999E+09,8.999999E+09,8.999999E+09]];
	LOCAL CONST Robtarget Tr_meulage_bavure_P7 :=[[-253.8703125,28.20916796875,16],[0.585429038982807,-0.60991227779775,0.385331857079332,-0.369863777122091],[0,0,0,0],[8.999999E+09,8.999999E+09,8.999999E+09,8.999999E+09,8.999999E+09,8.999999E+09]];
	LOCAL CONST Robtarget Tr_meulage_bavure_P8 :=[[-254.291984375,29.15475390625,16],[0.571032565854766,-0.598917795366762,0.40634773622671,-0.38742844550932],[0,0,0,0],[8.999999E+09,8.999999E+09,8.999999E+09,8.999999E+09,8.999999E+09,8.999999E+09]];
	LOCAL CONST Robtarget Tr_meulage_bavure_P9 :=[[-255.252375,31.292724609375,16],[0.553070298463584,-0.584255221402235,0.431329061913639,-0.408306651391239],[0,0,0,0],[8.999999E+09,8.999999E+09,8.999999E+09,8.999999E+09,8.999999E+09,8.999999E+09]];
	LOCAL CONST Robtarget Tr_meulage_bavure_P10 :=[[-255.56415625,32.53567578125,16],[0.531253682212153,-0.565456993391244,0.459799154321126,-0.431986864900475],[0,0,0,0],[8.999999E+09,8.999999E+09,8.999999E+09,8.999999E+09,8.999999E+09,8.999999E+09]];
	LOCAL CONST Robtarget Tr_meulage_bavure_P11 :=[[-255.7218125,33.414765625,16],[0.505827457095695,-0.542610762172791,0.490524548882518,-0.45727214147154],[0,0,0,0],[8.999999E+09,8.999999E+09,8.999999E+09,8.999999E+09,8.999999E+09,8.999999E+09]];
	LOCAL CONST Robtarget Tr_meulage_bavure_P12 :=[[-255.921,34.0666484375,16],[0.477580997210394,-0.516391764757695,0.52184884210419,-0.482627933700979],[0,0,0,0],[8.999999E+09,8.999999E+09,8.999999E+09,8.999999E+09,8.999999E+09,8.999999E+09]];
	LOCAL CONST Robtarget Tr_meulage_bavure_P13 :=[[-255.828,34.67721484375,16],[0.44771495152111,-0.487972263443213,0.552112218132097,-0.506563412500166],[0,0,0,0],[8.999999E+09,8.999999E+09,8.999999E+09,8.999999E+09,8.999999E+09,8.999999E+09]];
	LOCAL CONST Robtarget Tr_meulage_bavure_P14 :=[[-255.70228125,36.3830546875,16],[0.417684337405523,-0.458858628142605,0.579930030091689,-0.52789176339762],[0,0,0,0],[8.999999E+09,8.999999E+09,8.999999E+09,8.999999E+09,8.999999E+09,8.999999E+09]];
	LOCAL CONST Robtarget Tr_meulage_bavure_P15 :=[[-255.100484375,38.445890625,16],[0.388997912109695,-0.430686495468137,0.604348604515245,-0.54585028278471],[0,0,0,0],[8.999999E+09,8.999999E+09,8.999999E+09,8.999999E+09,8.999999E+09,8.999999E+09]];
	LOCAL CONST Robtarget Tr_meulage_bavure_P16 :=[[-254.95034375,38.88592578125,16],[0.362956420086452,-0.404912193743937,0.624918186046732,-0.560166058614374],[0,0,0,0],[8.999999E+09,8.999999E+09,8.999999E+09,8.999999E+09,8.999999E+09,8.999999E+09]];
	LOCAL CONST Robtarget Tr_meulage_bavure_P17 :=[[-254.361578125,39.786375,16],[0.340291841939914,-0.382411035867165,0.641751209164476,-0.571067988502311],[0,0,0,0],[8.999999E+09,8.999999E+09,8.999999E+09,8.999999E+09,8.999999E+09,8.999999E+09]];
	LOCAL CONST Robtarget Tr_meulage_bavure_P18 :=[[-252.592859375,42.4651796875,16],[0.320918216460952,-0.363167261242377,0.655465298133579,-0.579211776164721],[0,0,0,0],[8.999999E+09,8.999999E+09,8.999999E+09,8.999999E+09,8.999999E+09,8.999999E+09]];
	LOCAL CONST Robtarget Tr_meulage_bavure_P19 :=[[-251.71571875,43.65680078125,16],[0.304046866855106,-0.346358968008532,0.666945444769022,-0.585469676189562],[0,0,0,0],[8.999999E+09,8.999999E+09,8.999999E+09,8.999999E+09,8.999999E+09,8.999999E+09]];
	LOCAL CONST Robtarget Tr_meulage_bavure_P20 :=[[-250.668453125,44.9103984375,16],[0.288492305734553,-0.330689028543642,0.677110729198127,-0.590709756426627],[0,0,0,0],[8.999999E+09,8.999999E+09,8.999999E+09,8.999999E+09,8.999999E+09,8.999999E+09]];
	LOCAL CONST Robtarget Tr_meulage_bavure_P21 :=[[-249.75471875,45.80035546875,16],[0.273213722789649,-0.314985836579256,0.686618133293036,-0.595561687373419],[0,0,0,0],[8.999999E+09,8.999999E+09,8.999999E+09,8.999999E+09,8.999999E+09,8.999999E+09]];
	LOCAL CONST Robtarget Tr_meulage_bavure_P22 :=[[-248.145796875,47.2981875,16],[0.257669595136235,-0.298636902525126,0.695744494715929,-0.600301572765726],[0,0,0,0],[8.999999E+09,8.999999E+09,8.999999E+09,8.999999E+09,8.999999E+09,8.999999E+09]];
	LOCAL CONST Robtarget Tr_meulage_bavure_P23 :=[[-245.80265625,49.0953359375,16],[0.241989922027217,-0.281814881859191,0.704395878371599,-0.604853450459742],[0,0,0,0],[8.999999E+09,8.999999E+09,8.999999E+09,8.999999E+09,8.999999E+09,8.999999E+09]];
	LOCAL CONST Robtarget Tr_meulage_bavure_P24 :=[[-244.587734375,50.067140625,16],[0.226961967880884,-0.265447208154834,0.712193995689482,-0.608938221269031],[0,0,0,0],[8.999999E+09,8.999999E+09,8.999999E+09,8.999999E+09,8.999999E+09,8.999999E+09]];
	LOCAL CONST Robtarget Tr_meulage_bavure_P25 :=[[-243.97409375,50.5550234375,16],[0.213480402833133,-0.250614149302889,0.718816299364153,-0.612308577062103],[0,0,0,0],[8.999999E+09,8.999999E+09,8.999999E+09,8.999999E+09,8.999999E+09,8.999999E+09]];
	LOCAL CONST Robtarget Tr_meulage_bavure_P26 :=[[-241.878078125,52.121125,16],[0.202437374629555,-0.238413630201259,0.724034151414614,-0.614778494966008],[0,0,0,0],[8.999999E+09,8.999999E+09,8.999999E+09,8.999999E+09,8.999999E+09,8.999999E+09]];
	LOCAL CONST Robtarget Tr_meulage_bavure_P27 :=[[-238.73284375,54.03433203125,16],[0.194466247672732,-0.229637650602663,0.727757639209837,-0.616293961120423],[0,0,0,0],[8.999999E+09,8.999999E+09,8.999999E+09,8.999999E+09,8.999999E+09,8.999999E+09]];
	LOCAL CONST Robtarget Tr_meulage_bavure_P28 :=[[-235.927125,55.7035234375,16],[0.189778571349175,-0.224581578245878,0.73004581666173,-0.616911917654348],[0,0,0,0],[8.999999E+09,8.999999E+09,8.999999E+09,8.999999E+09,8.999999E+09,8.999999E+09]];
	LOCAL CONST Robtarget Tr_meulage_bavure_P29 :=[[-235.201171875,56.117828125,16],[0.188146156999226,-0.223008366759042,0.731062944857985,-0.616778130787286],[0,0,0,0],[8.999999E+09,8.999999E+09,8.999999E+09,8.999999E+09,8.999999E+09,8.999999E+09]];
	LOCAL CONST Robtarget Tr_meulage_bavure_P30 :=[[-232.130359375,57.76513671875,16],[0.188601133982388,-0.223795707366468,0.731190767551263,-0.616202203073549],[0,0,0,0],[8.999999E+09,8.999999E+09,8.999999E+09,8.999999E+09,8.999999E+09,8.999999E+09]];
	LOCAL CONST Robtarget Tr_meulage_bavure_P31 :=[[-232.333796875,57.77191015625,16],[0.189431852479978,-0.224924485000838,0.731055635090883,-0.615696522415855],[0,0,0,0],[8.999999E+09,8.999999E+09,8.999999E+09,8.999999E+09,8.999999E+09,8.999999E+09]];
	LOCAL CONST Robtarget Tr_meulage_bavure_P32 :=[[-226.89703125,60.77880859375,16],[0.188563245098339,-0.223935812796697,0.731422356330549,-0.615887969524437],[0,0,0,0],[8.999999E+09,8.999999E+09,8.999999E+09,8.999999E+09,8.999999E+09,8.999999E+09]];
	LOCAL CONST Robtarget Tr_meulage_bavure_P33 :=[[-225.39246875,61.7685546875,16],[0.184740660004619,-0.21934778881877,0.732738306249277,-0.617132085242952],[0,0,0,0],[8.999999E+09,8.999999E+09,8.999999E+09,8.999999E+09,8.999999E+09,8.999999E+09]];
	LOCAL CONST Robtarget Tr_meulage_bavure_P34 :=[[-224.47215625,62.27615234375,16],[0.178385071531956,-0.211678612554078,0.73479857525512,-0.61922692532283],[0,0,0,0],[8.999999E+09,8.999999E+09,8.999999E+09,8.999999E+09,8.999999E+09,8.999999E+09]];
	LOCAL CONST Robtarget Tr_meulage_bavure_P35 :=[[-221.91540625,63.70614453125,16],[0.170971436783367,-0.20269511296879,0.737024764035191,-0.621673512530228],[0,0,0,0],[8.999999E+09,8.999999E+09,8.999999E+09,8.999999E+09,8.999999E+09,8.999999E+09]];
	LOCAL CONST Robtarget Tr_meulage_bavure_P36 :=[[-218.78690625,65.289796875,16],[0.163857270059806,-0.194028044178679,0.738959483876873,-0.624053518785986],[0,0,0,0],[8.999999E+09,8.999999E+09,8.999999E+09,8.999999E+09,8.999999E+09,8.999999E+09]];
	LOCAL CONST Robtarget Tr_meulage_bavure_P37 :=[[-218.390453125,65.4821796875,16],[0.157793225459908,-0.186578582255451,0.740402915201095,-0.626173501359028],[0,0,0,0],[8.999999E+09,8.999999E+09,8.999999E+09,8.999999E+09,8.999999E+09,8.999999E+09]];
	LOCAL CONST Robtarget Tr_meulage_bavure_P38 :=[[-217.865296875,65.7450546875,16],[0.152937387192278,-0.180538308732001,0.74135699824237,-0.628017416825402],[0,0,0,0],[8.999999E+09,8.999999E+09,8.999999E+09,8.999999E+09,8.999999E+09,8.999999E+09]];
	LOCAL CONST Robtarget Tr_meulage_bavure_P39 :=[[-212.66384375,68.3941015625,16],[0.149169691487392,-0.175766968605694,0.741899540679204,-0.629634375990311],[0,0,0,0],[8.999999E+09,8.999999E+09,8.999999E+09,8.999999E+09,8.999999E+09,8.999999E+09]];
	LOCAL CONST Robtarget Tr_meulage_bavure_P40 :=[[-209.43584375,69.988765625,16],[0.146251184250401,-0.171985972516812,0.74213350424032,-0.631085793095348],[0,0,0,0],[8.999999E+09,8.999999E+09,8.999999E+09,8.999999E+09,8.999999E+09,8.999999E+09]];
	LOCAL CONST Robtarget Tr_meulage_bavure_P41 :=[[-207.854359375,70.7095,16],[0.143924493838873,-0.168890132501514,0.742145994321991,-0.632440658345641],[0,0,0,0],[8.999999E+09,8.999999E+09,8.999999E+09,8.999999E+09,8.999999E+09,8.999999E+09]];
	LOCAL CONST Robtarget Tr_meulage_bavure_P42 :=[[-205.927609375,71.6823125,16],[0.141950547609574,-0.166196035145421,0.742008383630811,-0.633760584571867],[0,0,0,0],[8.999999E+09,8.999999E+09,8.999999E+09,8.999999E+09,8.999999E+09,8.999999E+09]];
	LOCAL CONST Robtarget Tr_meulage_bavure_P43 :=[[-205.370859375,71.9528828125,16],[0.140068999219531,-0.163603532208807,0.741802462752603,-0.635093430890774],[0,0,0,0],[8.999999E+09,8.999999E+09,8.999999E+09,8.999999E+09,8.999999E+09,8.999999E+09]];
	LOCAL CONST Robtarget Tr_meulage_bavure_P44 :=[[-202.7099375,73.26184375,16],[0.138159275058758,-0.160967663765225,0.741551427011894,-0.636476949334245],[0,0,0,0],[8.999999E+09,8.999999E+09,8.999999E+09,8.999999E+09,8.999999E+09,8.999999E+09]];
	LOCAL CONST Robtarget Tr_meulage_bavure_P45 :=[[-198.0714375,75.5464453125,16],[0.136237911398741,-0.158308216330066,0.74124897370158,-0.637908848603354],[0,0,0,0],[8.999999E+09,8.999999E+09,8.999999E+09,8.999999E+09,8.999999E+09,8.999999E+09]];
	LOCAL CONST Robtarget Tr_meulage_bavure_P46 :=[[-197.192484375,75.9072890625,16],[0.134438126674159,-0.155782274790662,0.740864933989794,-0.639357038392233],[0,0,0,0],[8.999999E+09,8.999999E+09,8.999999E+09,8.999999E+09,8.999999E+09,8.999999E+09]];
	LOCAL CONST Robtarget Tr_meulage_bavure_P47 :=[[-195.189171875,76.8489375,16],[0.132929341443141,-0.15358059061161,0.74035067051119,-0.640799248629797],[0,0,0,0],[8.999999E+09,8.999999E+09,8.999999E+09,8.999999E+09,8.999999E+09,8.999999E+09]];
	LOCAL CONST Robtarget Tr_meulage_bavure_P48 :=[[-187.792515625,79.6225859375,16],[0.131759348339266,-0.151756496959202,0.739698282326842,-0.642227289110797],[0,0,0,0],[8.999999E+09,8.999999E+09,8.999999E+09,8.999999E+09,8.999999E+09,8.999999E+09]];
	LOCAL CONST Robtarget Tr_meulage_bavure_P49 :=[[-186.904734375,80.012359375,16],[0.130789351779827,-0.150146664223683,0.738940676049924,-0.643674453402024],[0,0,0,0],[8.999999E+09,8.999999E+09,8.999999E+09,8.999999E+09,8.999999E+09,8.999999E+09]];
	LOCAL CONST Robtarget Tr_meulage_bavure_P50 :=[[-185.277125,80.6110234375,16],[0.129744629435329,-0.148435880732408,0.73814354801645,-0.645195492053045],[0,0,0,0],[8.999999E+09,8.999999E+09,8.999999E+09,8.999999E+09,8.999999E+09,8.999999E+09]];
	LOCAL CONST Robtarget Tr_meulage_bavure_P51 :=[[-182.14228125,81.952609375,16],[0.12835161150222,-0.146317306553604,0.737374497622152,-0.646835342173076],[0,0,0,0],[8.999999E+09,8.999999E+09,8.999999E+09,8.999999E+09,8.999999E+09,8.999999E+09]];
	LOCAL CONST Robtarget Tr_meulage_bavure_P52 :=[[-182.051359375,81.9865078125,16],[0.126488661797153,-0.143657730278459,0.736655593170886,-0.64861514938988],[0,0,0,0],[8.999999E+09,8.999999E+09,8.999999E+09,8.999999E+09,8.999999E+09,8.999999E+09]];
	LOCAL CONST Robtarget Tr_meulage_bavure_P53 :=[[-181.98765625,82.0165078125,16],[0.124245754248217,-0.140571958200415,0.735973378563832,-0.650496505113079],[0,0,0,0],[8.999999E+09,8.999999E+09,8.999999E+09,8.999999E+09,8.999999E+09,8.999999E+09]];
	LOCAL CONST Robtarget Tr_meulage_bavure_P54 :=[[-178.7385625,83.323453125,16],[0.121890077248597,-0.13737159001805,0.735275955169324,-0.652411775701575],[0,0,0,0],[8.999999E+09,8.999999E+09,8.999999E+09,8.999999E+09,8.999999E+09,8.999999E+09]];
	LOCAL CONST Robtarget Tr_meulage_bavure_P55 :=[[-176.177203125,84.2620546875,16],[0.119744077520131,-0.134425526366505,0.734506708346704,-0.654286656713731],[0,0,0,0],[8.999999E+09,8.999999E+09,8.999999E+09,8.999999E+09,8.999999E+09,8.999999E+09]];
	LOCAL CONST Robtarget Tr_meulage_bavure_P56 :=[[-174.720828125,84.77596875,16],[0.118034676835162,-0.131992568389532,0.733641605599346,-0.656060798621567],[0,0,0,0],[8.999999E+09,8.999999E+09,8.999999E+09,8.999999E+09,8.999999E+09,8.999999E+09]];
	LOCAL CONST Robtarget Tr_meulage_bavure_P57 :=[[-167.2675,87.4896875,16],[0.116818783983896,-0.130134486232051,0.73268590280222,-0.657715557848938],[0,0,0,0],[8.999999E+09,8.999999E+09,8.999999E+09,8.999999E+09,8.999999E+09,8.999999E+09]];
	LOCAL CONST Robtarget Tr_meulage_bavure_P58 :=[[-165.52871875,88.1170078125,16],[0.115960119380232,-0.128701302114255,0.731691137098542,-0.659255114078654],[0,0,0,0],[8.999999E+09,8.999999E+09,8.999999E+09,8.999999E+09,8.999999E+09,8.999999E+09]];
	LOCAL CONST Robtarget Tr_meulage_bavure_P59 :=[[-161.09190625,89.690609375,16],[0.115180194483959,-0.127387658249532,0.730733344691187,-0.660707716226145],[0,0,0,0],[8.999999E+09,8.999999E+09,8.999999E+09,8.999999E+09,8.999999E+09,8.999999E+09]];
	LOCAL CONST Robtarget Tr_meulage_bavure_P60 :=[[-160.70334375,89.7634921875,16],[0.114172151383682,-0.125857457734846,0.729881884131689,-0.662115590661721],[0,0,0,0],[8.999999E+09,8.999999E+09,8.999999E+09,8.999999E+09,8.999999E+09,8.999999E+09]];
	LOCAL CONST Robtarget Tr_meulage_bavure_P61 :=[[-152.83928125,92.6495078125,16],[0.112698515167588,-0.123858070575124,0.729197790746435,-0.663497403915755],[0,0,0,0],[8.999999E+09,8.999999E+09,8.999999E+09,8.999999E+09,8.999999E+09,8.999999E+09]];
	LOCAL CONST Robtarget Tr_meulage_bavure_P62 :=[[-151.02440625,93.409578125,16],[0.110670370474892,-0.121297619700742,0.728700461210798,-0.664856822470112],[0,0,0,0],[8.999999E+09,8.999999E+09,8.999999E+09,8.999999E+09,8.999999E+09,8.999999E+09]];
	LOCAL CONST Robtarget Tr_meulage_bavure_P63 :=[[-149.873609375,93.77353125,16],[0.108155754336413,-0.11825943440918,0.728389036115191,-0.666157977543109],[0,0,0,0],[8.999999E+09,8.999999E+09,8.999999E+09,8.999999E+09,8.999999E+09,8.999999E+09]];
	LOCAL CONST Robtarget Tr_meulage_bavure_P64 :=[[-141.862515625,96.539796875,16],[0.105343724576514,-0.114951930797488,0.728229561545609,-0.667360816192686],[0,0,0,0],[8.999999E+09,8.999999E+09,8.999999E+09,8.999999E+09,8.999999E+09,8.999999E+09]];
	LOCAL CONST Robtarget Tr_meulage_bavure_P65 :=[[-140.6874375,96.9318515625,16],[0.102462919316256,-0.111622109033768,0.728179436536924,-0.668428427840118],[0,0,0,0],[8.999999E+09,8.999999E+09,8.999999E+09,8.999999E+09,8.999999E+09,8.999999E+09]];
	LOCAL CONST Robtarget Tr_meulage_bavure_P66 :=[[-140.123109375,97.0985078125,16],[0.0996901471133661,-0.108461282578978,0.728216797063141,-0.669326767151097],[0,0,0,0],[8.999999E+09,8.999999E+09,8.999999E+09,8.999999E+09,8.999999E+09,8.999999E+09]];
	LOCAL CONST Robtarget Tr_meulage_bavure_P67 :=[[-136.734890625,98.1063828125,16],[0.0971139193367168,-0.105560912596481,0.728328352074265,-0.670047455011692],[0,0,0,0],[8.999999E+09,8.999999E+09,8.999999E+09,8.999999E+09,8.999999E+09,8.999999E+09]];
	LOCAL CONST Robtarget Tr_meulage_bavure_P68 :=[[-134.11696875,99.0388203125,16],[0.0947425953279012,-0.102922912845174,0.728505843739634,-0.670604168104555],[0,0,0,0],[8.999999E+09,8.999999E+09,8.999999E+09,8.999999E+09,8.999999E+09,8.999999E+09]];
	LOCAL CONST Robtarget Tr_meulage_bavure_P69 :=[[-131.930234375,99.66159375,16],[0.0925589919612516,-0.100525656609279,0.728755398093229,-0.671001486675231],[0,0,0,0],[8.999999E+09,8.999999E+09,8.999999E+09,8.999999E+09,8.999999E+09,8.999999E+09]];
	LOCAL CONST Robtarget Tr_meulage_bavure_P70 :=[[-126.72521875,101.24625,16],[0.090591038674018,-0.0983925967020574,0.729061262585889,-0.671253928124713],[0,0,0,0],[8.999999E+09,8.999999E+09,8.999999E+09,8.999999E+09,8.999999E+09,8.999999E+09]];
	LOCAL CONST Robtarget Tr_meulage_bavure_P71 :=[[-122.15609375,102.54284375,16],[0.0889338386667942,-0.0966233476907753,0.729405915739793,-0.671358109435501],[0,0,0,0],[8.999999E+09,8.999999E+09,8.999999E+09,8.999999E+09,8.999999E+09,8.999999E+09]];
	LOCAL CONST Robtarget Tr_meulage_bavure_P72 :=[[-118.1851171875,103.655765625,16],[0.0877076022776948,-0.095344466798773,0.72976473898446,-0.67131232290827],[0,0,0,0],[8.999999E+09,8.999999E+09,8.999999E+09,8.999999E+09,8.999999E+09,8.999999E+09]];
	LOCAL CONST Robtarget Tr_meulage_bavure_P73 :=[[-115.516875,104.3459140625,16],[0.0869805222386408,-0.0946260832761608,0.730117111070816,-0.671125396059866],[0,0,0,0],[8.999999E+09,8.999999E+09,8.999999E+09,8.999999E+09,8.999999E+09,8.999999E+09]];
	LOCAL CONST Robtarget Tr_meulage_bavure_P74 :=[[-114.05465625,104.7516796875,16],[0.0866722053443163,-0.0943778930219965,0.730463507233294,-0.670823230612892],[0,0,0,0],[8.999999E+09,8.999999E+09,8.999999E+09,8.999999E+09,8.999999E+09,8.999999E+09]];
	LOCAL CONST Robtarget Tr_meulage_bavure_P75 :=[[-111.3724375,105.4299296875,16],[0.0865133873679466,-0.0943034340892468,0.730828008508422,-0.670457096393731],[0,0,0,0],[8.999999E+09,8.999999E+09,8.999999E+09,8.999999E+09,8.999999E+09,8.999999E+09]];
	LOCAL CONST Robtarget Tr_meulage_bavure_P76 :=[[-107.8739296875,106.2517109375,16],[0.0860988791706962,-0.0939587304139098,0.731259602656315,-0.670088153534656],[0,0,0,0],[8.999999E+09,8.999999E+09,8.999999E+09,8.999999E+09,8.999999E+09,8.999999E+09]];
	LOCAL CONST Robtarget Tr_meulage_bavure_P77 :=[[-105.351015625,106.9495234375,16],[0.0850180313960092,-0.0928894208649515,0.731798747672506,-0.669786594919511],[0,0,0,0],[8.999999E+09,8.999999E+09,8.999999E+09,8.999999E+09,8.999999E+09,8.999999E+09]];
	LOCAL CONST Robtarget Tr_meulage_bavure_P78 :=[[-100.3968828125,108.125671875,16],[0.0830226033403211,-0.0908163324771312,0.73245853586199,-0.669599980834012],[0,0,0,0],[8.999999E+09,8.999999E+09,8.999999E+09,8.999999E+09,8.999999E+09,8.999999E+09]];
	LOCAL CONST Robtarget Tr_meulage_bavure_P79 :=[[-98.9347265625,108.560578125,16],[0.0801269017929764,-0.0877495923262772,0.733221060322284,-0.669527120701989],[0,0,0,0],[8.999999E+09,8.999999E+09,8.999999E+09,8.999999E+09,8.999999E+09,8.999999E+09]];
	LOCAL CONST Robtarget Tr_meulage_bavure_P80 :=[[-94.913328125,109.371859375,16],[0.0765828575088332,-0.0839578583698632,0.734025097247842,-0.669547086144076],[0,0,0,0],[8.999999E+09,8.999999E+09,8.999999E+09,8.999999E+09,8.999999E+09,8.999999E+09]];
	LOCAL CONST Robtarget Tr_meulage_bavure_P81 :=[[-90.4933203125,110.2268046875,16],[0.0727539765233362,-0.079836158089158,0.734805772521754,-0.66962192573893],[0,0,0,0],[8.999999E+09,8.999999E+09,8.999999E+09,8.999999E+09,8.999999E+09,8.999999E+09]];
	LOCAL CONST Robtarget Tr_meulage_bavure_P82 :=[[-89.344234375,110.51171875,16],[0.0689348678767823,-0.0757061625975068,0.735513890784173,-0.669728211589671],[0,0,0,0],[8.999999E+09,8.999999E+09,8.999999E+09,8.999999E+09,8.999999E+09,8.999999E+09]];
	LOCAL CONST Robtarget Tr_meulage_bavure_P83 :=[[-88.2133515625,110.6929609375,16],[0.0652228586037968,-0.0716746809388804,0.736129834774758,-0.66986684138144],[0,0,0,0],[8.999999E+09,8.999999E+09,8.999999E+09,8.999999E+09,8.999999E+09,8.999999E+09]];
	LOCAL CONST Robtarget Tr_meulage_bavure_P84 :=[[-84.75,111.4052109375,16],[0.0615541117848836,-0.0676712615515534,0.736649053976782,-0.67005959657146],[0,0,0,0],[8.999999E+09,8.999999E+09,8.999999E+09,8.999999E+09,8.999999E+09,8.999999E+09]];
	LOCAL CONST Robtarget Tr_meulage_bavure_P85 :=[[-82.0062265625,112.0165390625,16],[0.0578257214064526,-0.0635843747848279,0.737076644180516,-0.670321739040764],[0,0,0,0],[8.999999E+09,8.999999E+09,8.999999E+09,8.999999E+09,8.999999E+09,8.999999E+09]];
	LOCAL CONST Robtarget Tr_meulage_bavure_P86 :=[[-79.32821875,112.50665625,16],[0.0540528838848583,-0.0594330372769014,0.737407292517104,-0.670653774138613],[0,0,0,0],[8.999999E+09,8.999999E+09,8.999999E+09,8.999999E+09,8.999999E+09,8.999999E+09]];
	LOCAL CONST Robtarget Tr_meulage_bavure_P87 :=[[-75.7334921875,113.099453125,16],[0.0504254805034586,-0.055427741066029,0.737617137625861,-0.671048429486982],[0,0,0,0],[8.999999E+09,8.999999E+09,8.999999E+09,8.999999E+09,8.999999E+09,8.999999E+09]];
	LOCAL CONST Robtarget Tr_meulage_bavure_P88 :=[[-73.439453125,113.5042109375,16],[0.0472450714580366,-0.0519021321768341,0.73768146268102,-0.671490976495749],[0,0,0,0],[8.999999E+09,8.999999E+09,8.999999E+09,8.999999E+09,8.999999E+09,8.999999E+09]];
	LOCAL CONST Robtarget Tr_meulage_bavure_P89 :=[[-72.397734375,113.57559375,16],[0.0447684120225403,-0.049140963567394,0.737594628375828,-0.671963629354872],[0,0,0,0],[8.999999E+09,8.999999E+09,8.999999E+09,8.999999E+09,8.999999E+09,8.999999E+09]];
	LOCAL CONST Robtarget Tr_meulage_bavure_P90 :=[[-64.626953125,114.6755078125,16],[0.043074126369996,-0.0472306330834042,0.737359824750743,-0.672468866029912],[0,0,0,0],[8.999999E+09,8.999999E+09,8.999999E+09,8.999999E+09,8.999999E+09,8.999999E+09]];
	LOCAL CONST Robtarget Tr_meulage_bavure_P91 :=[[-62.00521875,115.033078125,16],[0.0420633438952746,-0.0460622063612357,0.736995190461685,-0.673013400670319],[0,0,0,0],[8.999999E+09,8.999999E+09,8.999999E+09,8.999999E+09,8.999999E+09,8.999999E+09]];
	LOCAL CONST Robtarget Tr_meulage_bavure_P92 :=[[-59.59191796875,115.384640625,16],[0.0415295907279451,-0.0454085987883709,0.736523869762909,-0.673606666771875],[0,0,0,0],[8.999999E+09,8.999999E+09,8.999999E+09,8.999999E+09,8.999999E+09,8.999999E+09]];
	LOCAL CONST Robtarget Tr_meulage_bavure_P93 :=[[-53.6976015625,116.051546875,16],[0.0412672531593628,-0.0450445712639092,0.735969395343102,-0.67425295663767],[0,0,0,0],[8.999999E+09,8.999999E+09,8.999999E+09,8.999999E+09,8.999999E+09,8.999999E+09]];
	LOCAL CONST Robtarget Tr_meulage_bavure_P94 :=[[-53.68115234375,116.05353125,16],[0.0411039435307525,-0.0447826782825847,0.735356055313467,-0.674949219916489],[0,0,0,0],[8.999999E+09,8.999999E+09,8.999999E+09,8.999999E+09,8.999999E+09,8.999999E+09]];
	LOCAL CONST Robtarget Tr_meulage_bavure_P95 :=[[-53.6552734375,116.0562421875,16],[0.0408624366324264,-0.0444303637839806,0.734700201959521,-0.675700982156399],[0,0,0,0],[8.999999E+09,8.999999E+09,8.999999E+09,8.999999E+09,8.999999E+09,8.999999E+09]];
	LOCAL CONST Robtarget Tr_meulage_bavure_P96 :=[[-45.012390625,116.964296875,16],[0.0403235812553287,-0.0437520386100116,0.734027466328646,-0.676508275328072],[0,0,0,0],[8.999999E+09,8.999999E+09,8.999999E+09,8.999999E+09,8.999999E+09,8.999999E+09]];
	LOCAL CONST Robtarget Tr_meulage_bavure_P97 :=[[-43.1705625,117.17315625,16],[0.0392428653151048,-0.0424868254527491,0.733364689877086,-0.677370724807541],[0,0,0,0],[8.999999E+09,8.999999E+09,8.999999E+09,8.999999E+09,8.999999E+09,8.999999E+09]];
	LOCAL CONST Robtarget Tr_meulage_bavure_P98 :=[[-41.9234921875,117.3466171875,16],[0.0374335486933903,-0.0404379214857073,0.732726829162997,-0.678288211428501],[0,0,0,0],[8.999999E+09,8.999999E+09,8.999999E+09,8.999999E+09,8.999999E+09,8.999999E+09]];
	LOCAL CONST Robtarget Tr_meulage_bavure_P99 :=[[-40.4229140625,117.44128125,16],[0.0348811265492393,-0.0375965155591936,0.732119650917831,-0.679242685472885],[0,0,0,0],[8.999999E+09,8.999999E+09,8.999999E+09,8.999999E+09,8.999999E+09,8.999999E+09]];
	LOCAL CONST Robtarget Tr_meulage_bavure_P100 :=[[-33.30901953125,117.9559296875,16],[0.0317753527511481,-0.0341731716308694,0.731534783112439,-0.680205397210919],[0,0,0,0],[8.999999E+09,8.999999E+09,8.999999E+09,8.999999E+09,8.999999E+09,8.999999E+09]];
	LOCAL CONST Robtarget Tr_meulage_bavure_P101 :=[[-31.98034765625,118.085171875,16],[0.0284313083369646,-0.0305099826494235,0.730952934988928,-0.681152412090021],[0,0,0,0],[8.999999E+09,8.999999E+09,8.999999E+09,8.999999E+09,8.999999E+09,8.999999E+09]];
	LOCAL CONST Robtarget Tr_meulage_bavure_P102 :=[[-27.466064453125,118.5026875,16],[0.0251630064701749,-0.0269457175224156,0.730373402884623,-0.68205237612028],[0,0,0,0],[8.999999E+09,8.999999E+09,8.999999E+09,8.999999E+09,8.999999E+09,8.999999E+09]];
	LOCAL CONST Robtarget Tr_meulage_bavure_P103 :=[[-23.450255859375,118.6833515625,16],[0.0221483305238203,-0.0236695979960457,0.729798354191542,-0.682893523036373],[0,0,0,0],[8.999999E+09,8.999999E+09,8.999999E+09,8.999999E+09,8.999999E+09,8.999999E+09]];
	LOCAL CONST Robtarget Tr_meulage_bavure_P104 :=[[-15.8180234375,119.0326875,16],[0.0193868321243504,-0.0206785380281567,0.729231706306384,-0.683679506291273],[0,0,0,0],[8.999999E+09,8.999999E+09,8.999999E+09,8.999999E+09,8.999999E+09,8.999999E+09]];
	LOCAL CONST Robtarget Tr_meulage_bavure_P105 :=[[-12.7677001953125,119.2099921875,16],[0.0167548014520303,-0.0178387386126664,0.728686874006833,-0.68440959642831],[0,0,0,0],[8.999999E+09,8.999999E+09,8.999999E+09,8.999999E+09,8.999999E+09,8.999999E+09]];
	LOCAL CONST Robtarget Tr_meulage_bavure_P106 :=[[-11.2499697265625,119.246609375,16],[0.0141016603585383,-0.0149885716190527,0.728172584842414,-0.68508479225558],[0,0,0,0],[8.999999E+09,8.999999E+09,8.999999E+09,8.999999E+09,8.999999E+09,8.999999E+09]];
	LOCAL CONST Robtarget Tr_meulage_bavure_P107 :=[[-6.74887109375,119.3916328125,16],[0.0113514539464575,-0.0120465879315752,0.727693443283651,-0.685702761270867],[0,0,0,0],[8.999999E+09,8.999999E+09,8.999999E+09,8.999999E+09,8.999999E+09,8.999999E+09]];
	LOCAL CONST Robtarget Tr_meulage_bavure_P108 :=[[-5.0588076171875,119.4722578125,16],[0.00854411446470486,-0.00905430881153603,0.727244516123833,-0.686265569125955],[0,0,0,0],[8.999999E+09,8.999999E+09,8.999999E+09,8.999999E+09,8.999999E+09,8.999999E+09]];
	LOCAL CONST Robtarget Tr_meulage_bavure_P109 :=[[-2.4659423828125,119.5382109375,16],[0.00578941701890455,-0.00612696100487176,0.726818963898168,-0.686777356002235],[0,0,0,0],[8.999999E+09,8.999999E+09,8.999999E+09,8.999999E+09,8.999999E+09,8.999999E+09]];
	LOCAL CONST Robtarget Tr_meulage_bavure_P110 :=[[4.02682495117188,119.56246875,16],[0.00321751468728298,-0.00340094713674738,0.726417531276489,-0.687237696442782],[0,0,0,0],[8.999999E+09,8.999999E+09,8.999999E+09,8.999999E+09,8.999999E+09,8.999999E+09]];
	LOCAL CONST Robtarget Tr_meulage_bavure_P111 :=[[5.3006591796875,119.5595390625,16],[0.00094644297954575,-0.000999263543398247,0.726034606895245,-0.68765678598304],[0,0,0,0],[8.999999E+09,8.999999E+09,8.999999E+09,8.999999E+09,8.999999E+09,8.999999E+09]];
	LOCAL CONST Robtarget Tr_meulage_bavure_P112 :=[[5.386322265625,119.5638125,16],[0.000942596962523084,-0.00099414517197246,-0.725669420966971,0.688042160524923],[0,0,0,0],[8.999999E+09,8.999999E+09,8.999999E+09,8.999999E+09,8.999999E+09,8.999999E+09]];
	LOCAL CONST Robtarget Tr_meulage_bavure_P113 :=[[5.67303466796875,119.5661640625,16],[0.00239560273216607,-0.00252404997790309,-0.725317068623358,0.688406159344088],[0,0,0,0],[8.999999E+09,8.999999E+09,8.999999E+09,8.999999E+09,8.999999E+09,8.999999E+09]];
	LOCAL CONST Robtarget Tr_meulage_bavure_P114 :=[[14.6903994140625,119.544890625,16],[0.00341724316013773,-0.00359688497309214,-0.724970136088528,0.688762431210832],[0,0,0,0],[8.999999E+09,8.999999E+09,8.999999E+09,8.999999E+09,8.999999E+09,8.999999E+09]];
	LOCAL CONST Robtarget Tr_meulage_bavure_P115 :=[[15.6702265625,119.4904453125,16],[0.00410958508705164,-0.00432130671146169,-0.72462272978296,0.68911997293694],[0,0,0,0],[8.999999E+09,8.999999E+09,8.999999E+09,8.999999E+09,8.999999E+09,8.999999E+09]];
	LOCAL CONST Robtarget Tr_meulage_bavure_P116 :=[[24.301849609375,119.0535546875,16],[0.00469739019183538,-0.00493429722386243,-0.72426335600874,0.689489795703496],[0,0,0,0],[8.999999E+09,8.999999E+09,8.999999E+09,8.999999E+09,8.999999E+09,8.999999E+09]];
	LOCAL CONST Robtarget Tr_meulage_bavure_P117 :=[[24.73959375,119.022828125,16],[0.00548537545723063,-0.00575573235764647,-0.723881000103257,0.689879032795337],[0,0,0,0],[8.999999E+09,8.999999E+09,8.999999E+09,8.999999E+09,8.999999E+09,8.999999E+09]];
	LOCAL CONST Robtarget Tr_meulage_bavure_P118 :=[[25.040130859375,119.025390625,16],[0.0067326167580162,-0.00705620468084419,-0.723467140161985,0.690289923838477],[0,0,0,0],[8.999999E+09,8.999999E+09,8.999999E+09,8.999999E+09,8.999999E+09,8.999999E+09]];
	LOCAL CONST Robtarget Tr_meulage_bavure_P119 :=[[25.782470703125,118.980625,16],[0.00855738048065719,-0.00895712666281872,-0.723001801709374,0.690735069217029],[0,0,0,0],[8.999999E+09,8.999999E+09,8.999999E+09,8.999999E+09,8.999999E+09,8.999999E+09]];
	LOCAL CONST Robtarget Tr_meulage_bavure_P120 :=[[29.3323671875,118.8803984375,16],[0.0108789189502222,-0.0113709729601926,-0.722478224557496,0.691214557960596],[0,0,0,0],[8.999999E+09,8.999999E+09,8.999999E+09,8.999999E+09,8.999999E+09,8.999999E+09]];
	LOCAL CONST Robtarget Tr_meulage_bavure_P121 :=[[35.4125078125,118.4643828125,16],[0.0134897112865089,-0.0140777737396653,-0.721889087693566,0.69173404502373],[0,0,0,0],[8.999999E+09,8.999999E+09,8.999999E+09,8.999999E+09,8.999999E+09,8.999999E+09]];
	LOCAL CONST Robtarget Tr_meulage_bavure_P122 :=[[35.8721015625,118.4392734375,16],[0.0161744868939734,-0.0168506907901504,-0.721237047649402,0.69229441807051],[0,0,0,0],[8.999999E+09,8.999999E+09,8.999999E+09,8.999999E+09,8.999999E+09,8.999999E+09]];
	LOCAL CONST Robtarget Tr_meulage_bavure_P123 :=[[35.96591015625,118.438109375,16],[0.018810623546686,-0.0195603990735073,-0.720520702397392,0.692902207130731],[0,0,0,0],[8.999999E+09,8.999999E+09,8.999999E+09,8.999999E+09,8.999999E+09,8.999999E+09]];
	LOCAL CONST Robtarget Tr_meulage_bavure_P124 :=[[36.19030859375,118.4218125,16],[0.0214076603885088,-0.0222153243131728,-0.719732433902051,0.693565725098769],[0,0,0,0],[8.999999E+09,8.999999E+09,8.999999E+09,8.999999E+09,8.999999E+09,8.999999E+09]];
	LOCAL CONST Robtarget Tr_meulage_bavure_P125 :=[[44.78408984375,117.97659375,16],[0.0240331469400272,-0.0248849284707739,-0.718879594587187,0.694273200310458],[0,0,0,0],[8.999999E+09,8.999999E+09,8.999999E+09,8.999999E+09,8.999999E+09,8.999999E+09]];
	LOCAL CONST Robtarget Tr_meulage_bavure_P126 :=[[46.3662421875,117.8996875,16],[0.0267363943141935,-0.0276191578507155,-0.717964790252599,0.695017199280877],[0,0,0,0],[8.999999E+09,8.999999E+09,8.999999E+09,8.999999E+09,8.999999E+09,8.999999E+09]];
	LOCAL CONST Robtarget Tr_meulage_bavure_P127 :=[[53.729859375,117.176296875,16],[0.0295107446481412,-0.0304094834885107,-0.71698731648897,0.695797073332607],[0,0,0,0],[8.999999E+09,8.999999E+09,8.999999E+09,8.999999E+09,8.999999E+09,8.999999E+09]];
	LOCAL CONST Robtarget Tr_meulage_bavure_P128 :=[[59.17199609375,116.7133515625,16],[0.032281126411846,-0.0331775635675912,-0.715954874211935,0.696610218303948],[0,0,0,0],[8.999999E+09,8.999999E+09,8.999999E+09,8.999999E+09,8.999999E+09,8.999999E+09]];
	LOCAL CONST Robtarget Tr_meulage_bavure_P129 :=[[65.04940625,115.9971953125,16],[0.0349685733366355,-0.035842620505372,-0.714882349536186,0.697449447455319],[0,0,0,0],[8.999999E+09,8.999999E+09,8.999999E+09,8.999999E+09,8.999999E+09,8.999999E+09]];
